REGION Network 2: Watchdog
   // Use S7 comm counter as a live count, but could be anything as long as its changing
   RUNG wire#powerrail
      #Watchdog(bEnable := true, nLocalCount := "S7_Internal_DB".CommCycles, nRemoteCount := "DB_ToHB".WatchdogCounter, sTag := "DB_Customer".Watchdog, bOk => #bWatchdogOk)
   END_RUNG
   // the same network as SCL:
   #Watchdog(bEnable := true,   // "fbHeartbeatCount2"
             nLocalCount := "S7_Internal_DB".CommCycles,
             nRemoteCount := "DB_ToHB".WatchdogCounter,
             sTag := "DB_Customer".Watchdog,
             bOk => #bWatchdogOk);
END_REGION

REGION Network 3: Start request
   RUNG wire#powerrail
      P_Contact(operand := "DB_ToHB".StartRequest, bit := #epStartRequest)
      Contact( "DB_ToHB".EnableHeatbooster )
      S_Coil( "DB_Application".ToHB.StartRequest )
   END_RUNG
   RUNG wire#powerrail
      N_Contact(operand := "DB_ToHB".StartRequest, bit := #enStartRequest)
      R_Coil( "DB_Application".ToHB.StartRequest )
   END_RUNG
   // the same network as SCL:
   #_w1 := "DB_ToHB".StartRequest AND NOT #epStartRequest;   // rising edge of "DB_ToHB".StartRequest
   #epStartRequest := "DB_ToHB".StartRequest;
   IF #_w1 AND "DB_ToHB".EnableHeatbooster THEN "DB_Application".ToHB.StartRequest := TRUE; END_IF;
   #_w2 := NOT "DB_ToHB".StartRequest AND #enStartRequest;   // falling edge of "DB_ToHB".StartRequest
   #enStartRequest := "DB_ToHB".StartRequest;
   IF #_w2 THEN "DB_Application".ToHB.StartRequest := FALSE; END_IF;
END_REGION

REGION Network 4: Stop request
   // a low enable signal is the same as a stop request
   // a watchdog timeout is the same as a stop request
   // a FastStoprequest is also a stop request
   RUNG wire#powerrail
      Contact( "DB_ToHB".StopRequest )
      wire#w1
      Coil( #bStopReq )
   END_RUNG
   RUNG wire#powerrail
      I_Contact( "DB_ToHB".EnableHeatbooster )
   END_RUNG wire#w1
   RUNG wire#powerrail
      I_Contact( #bWatchdogOk )
   END_RUNG wire#w1
   RUNG wire#powerrail
      Contact( "DB_ToHB".FastStopRequest )
   END_RUNG wire#w1
   RUNG wire#powerrail
      P_Contact(operand := #bStopReq, bit := #epStopRequest)
      S_Coil( "DB_Application".ToHB.StopRequest )
   END_RUNG
   RUNG wire#powerrail
      N_Contact(operand := #bStopReq, bit := #enStopRequest)
      R_Coil( "DB_Application".ToHB.StopRequest )
   END_RUNG
   // the same network as SCL:
   #bStopReq := "DB_ToHB".StopRequest OR NOT "DB_ToHB".EnableHeatbooster OR NOT #bWatchdogOk OR "DB_ToHB".FastStopRequest;
   #_w1 := #bStopReq AND NOT #epStopRequest;   // rising edge of #bStopReq
   #epStopRequest := #bStopReq;
   IF #_w1 THEN "DB_Application".ToHB.StopRequest := TRUE; END_IF;
   #_w2 := NOT #bStopReq AND #enStopRequest;   // falling edge of #bStopReq
   #enStopRequest := #bStopReq;
   IF #_w2 THEN "DB_Application".ToHB.StopRequest := FALSE; END_IF;
END_REGION

REGION Network 5: Commands
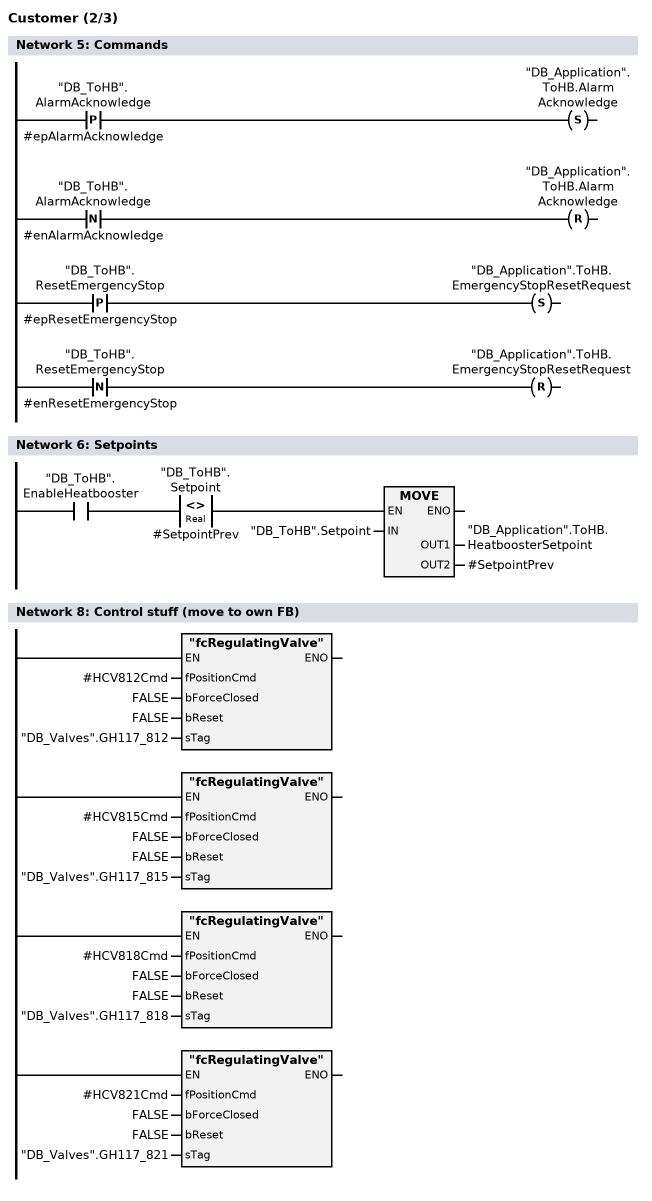
   RUNG wire#powerrail
      P_Contact(operand := "DB_ToHB".AlarmAcknowledge, bit := #epAlarmAcknowledge)
      S_Coil( "DB_Application".ToHB.AlarmAcknowledge )
   END_RUNG
   RUNG wire#powerrail
      N_Contact(operand := "DB_ToHB".AlarmAcknowledge, bit := #enAlarmAcknowledge)
      R_Coil( "DB_Application".ToHB.AlarmAcknowledge )
   END_RUNG
   RUNG wire#powerrail
      P_Contact(operand := "DB_ToHB".ResetEmergencyStop, bit := #epResetEmergencyStop)
      S_Coil( "DB_Application".ToHB.EmergencyStopResetRequest )
   END_RUNG
   RUNG wire#powerrail
      N_Contact(operand := "DB_ToHB".ResetEmergencyStop, bit := #enResetEmergencyStop)
      R_Coil( "DB_Application".ToHB.EmergencyStopResetRequest )
   END_RUNG
   // the same network as SCL:
   #_w1 := "DB_ToHB".AlarmAcknowledge AND NOT #epAlarmAcknowledge;   // rising edge of "DB_ToHB".AlarmAcknowledge
   #epAlarmAcknowledge := "DB_ToHB".AlarmAcknowledge;
   IF #_w1 THEN "DB_Application".ToHB.AlarmAcknowledge := TRUE; END_IF;
   #_w2 := NOT "DB_ToHB".AlarmAcknowledge AND #enAlarmAcknowledge;   // falling edge of "DB_ToHB".AlarmAcknowledge
   #enAlarmAcknowledge := "DB_ToHB".AlarmAcknowledge;
   IF #_w2 THEN "DB_Application".ToHB.AlarmAcknowledge := FALSE; END_IF;
   #_w3 := "DB_ToHB".ResetEmergencyStop AND NOT #epResetEmergencyStop;   // rising edge of "DB_ToHB".ResetEmergencyStop
   #epResetEmergencyStop := "DB_ToHB".ResetEmergencyStop;
   IF #_w3 THEN "DB_Application".ToHB.EmergencyStopResetRequest := TRUE; END_IF;
   #_w4 := NOT "DB_ToHB".ResetEmergencyStop AND #enResetEmergencyStop;   // falling edge of "DB_ToHB".ResetEmergencyStop
   #enResetEmergencyStop := "DB_ToHB".ResetEmergencyStop;
   IF #_w4 THEN "DB_Application".ToHB.EmergencyStopResetRequest := FALSE; END_IF;
END_REGION

REGION Network 6: Setpoints
   RUNG wire#powerrail
      Contact( "DB_ToHB".EnableHeatbooster )
      { S7_Templates := "SrcType := Real" } NE_Contact(in1 := "DB_ToHB".Setpoint, in2 := #SetpointPrev)
      Move(in := "DB_ToHB".Setpoint, out1 => "DB_Application".ToHB.HeatboosterSetpoint, out2 => #SetpointPrev)
   END_RUNG
   // the same network as SCL:
   IF "DB_ToHB".EnableHeatbooster AND ("DB_ToHB".Setpoint <> #SetpointPrev) THEN
       "DB_Application".ToHB.HeatboosterSetpoint := "DB_ToHB".Setpoint;
       #SetpointPrev := "DB_ToHB".Setpoint;
   END_IF;
END_REGION

REGION Network 7 (SCL): To Customer
   "DB_FromHB".CompressorMotorPower            := "DB_Heatbooster".Inverter.HBL_SC_10_A3.fValue;
   "DB_FromHB".CompressorMotorSpeed            := "DB_Heatbooster".Inverter.HBL_SC_10_A1.fValue;
   //"DB_FromHB".HBL_CT_524                      := "DB_Heatbooster".AI.HBL_CT_524.fValue;
   //"DB_FromHB".HBL_CT_538                      := "DB_Heatbooster".AI.HBL_CT_538.fValue;
   "DB_FromHB".HBL_CT_615    := "DB_Heatbooster".AI.HBL_TT_546.fValue;
   "DB_FromHB".HBL_CT_620  := "DB_Heatbooster".AI.HBL_TT_542.fValue;
   "DB_FromHB".HBL_SC_02_A3         := "DB_Heatbooster".AI.HBL_TT_16.fValue;
   "DB_FromHB".HBL_SC_10_A1    := "DB_Heatbooster".AI.HBL_TT_17.fValue;
   "DB_FromHB".HBL_SC_10_A2           := "DB_Heatbooster".AI.HBL_TT_18.fValue;

   "DB_FromHB".HBL_CT_643   := "DB_Heatbooster".AI.HBL_CT_01.fValue;
   "DB_FromHB".HBL_CT_673 := "DB_Heatbooster".AI.HBL_CT_615.fValue;
   "DB_FromHB".HBL_CT_950 := "DB_Heatbooster".AI.HBL_CT_03.fValue;
   "DB_FromHB".HBL_SC_10_A3 := "DB_Heatbooster".AI.SSC_LT_01.fValue;
   "DB_FromHB".TemperatureLift                 := "DB_Heatbooster".Calc.System.TemperatureLift.fValue;
   "DB_FromHB".COP                             := "DB_Heatbooster".Calc.System.COP.fValue;
   "DB_FromHB".HeatSinkHeatRate                := "DB_Heatbooster".Calc.HeatSink.HeatRate.fValue;
   "DB_FromHB".CompressorMotorPower := "DB_Heatbooster".Calc.System.ElectricalPower.fValue;
   "DB_FromHB".HeatboosterPerformance             := "DB_Application".FromHB.HeatboosterSetpoint;
   //"DB_FromHB".WatchdogCounter                := "DB_Application".FromHB.RegulationTarget;
   "DB_FromHB".RunningTimeHours                := INT_TO_UINT("DB_Application".FromHB.RunningTimeHours);
   "DB_FromHB".RunningTimeMinutes              := "DB_Application".FromHB.RunningTimeMinutes;
   "DB_FromHB".RunningTimeSeconds              := "DB_Application".FromHB.RunningTimeSeconds;

   "DB_FromHB".HeatboosterState                := "DB_Application".FromHB.MachineState;
   "DB_FromHB".EmergencyStopStatus             := "DB_Application".FromHB.EmergencyStop;
   "DB_FromHB".HBL_EC_01 := "DB_DO".HBL_EC_01;
   "DB_FromHB".HBL_EC_02 := "DB_DO".HBL_EC_02;
   "DB_FromHB".AlarmActive                    := "DB_DO".GH117_826_1;
   "DB_FromHB".WarningActive                    := "DB_DO".GH117_826_2;

   "DB_FromHB".Alarms                          := "DB_Application".FromHB.Alarms;
   //"DB_FromHB".HBL_SC_03_A1 := FALSE;
   //"DB_FromHB".HBL_SC_03_A2:= FALSE;
   //"DB_FromHB".HBL_SC_03_A3   := FALSE;
   //"DB_FromHB".HBL_SC_01_A1  := FALSE;
   //"DB_FromHB".HBL_SC_01_A2          := 0.0;
   "DB_FromHB".HBL_SC_01_A3            := 0.0;
   "DB_FromHB".HBL_SC_02_A1            := 0.0;
   "DB_FromHB".HBL_SC_02_A2              := 0.0;
   "DB_FromHB".WatchdogCounter                 := "DB_Customer".Watchdog.nLocalCount;
END_REGION

REGION Network 8: Control stuff (move to own FB)
   RUNG wire#powerrail
      "fcRegulatingValve"(fPositionCmd := #HCV812Cmd, bForceClosed := FALSE, bReset := FALSE, sTag := "DB_Valves".GH117_812)
   END_RUNG
   RUNG wire#powerrail
      "fcRegulatingValve"(fPositionCmd := #HCV815Cmd, bForceClosed := FALSE, bReset := FALSE, sTag := "DB_Valves".GH117_815)
   END_RUNG
   RUNG wire#powerrail
      "fcRegulatingValve"(fPositionCmd := #HCV818Cmd, bForceClosed := FALSE, bReset := FALSE, sTag := "DB_Valves".GH117_818)
   END_RUNG
   RUNG wire#powerrail
      "fcRegulatingValve"(fPositionCmd := #HCV821Cmd, bForceClosed := FALSE, bReset := FALSE, sTag := "DB_Valves".GH117_821)
   END_RUNG
   // the same network as SCL:
   "fcRegulatingValve"(fPositionCmd := #HCV812Cmd,
                       bForceClosed := FALSE,
                       bReset := FALSE,
                       sTag := "DB_Valves".GH117_812);
   "fcRegulatingValve"(fPositionCmd := #HCV815Cmd,
                       bForceClosed := FALSE,
                       bReset := FALSE,
                       sTag := "DB_Valves".GH117_815);
   "fcRegulatingValve"(fPositionCmd := #HCV818Cmd,
                       bForceClosed := FALSE,
                       bReset := FALSE,
                       sTag := "DB_Valves".GH117_818);
   "fcRegulatingValve"(fPositionCmd := #HCV821Cmd,
                       bForceClosed := FALSE,
                       bReset := FALSE,
                       sTag := "DB_Valves".GH117_821);
END_REGION

REGION Network 9: Analog outputs
   // Move to own FB in Section 30
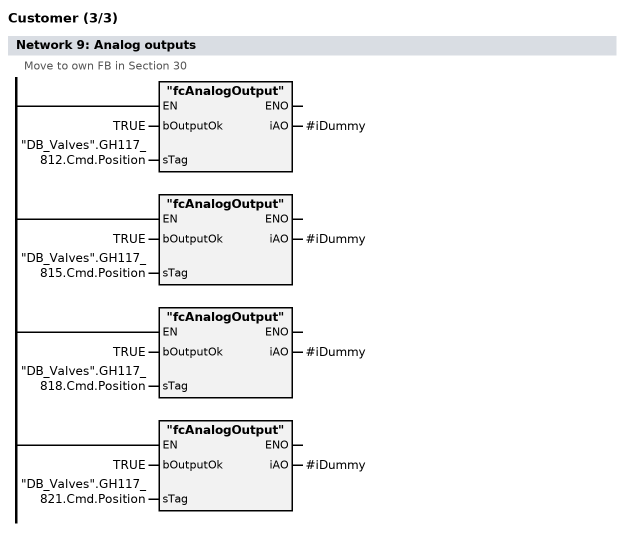
   RUNG wire#powerrail
      "fcAnalogOutput"(bOutputOk := TRUE, sTag := "DB_Valves".GH117_812.Cmd.Position, iAO => #iDummy)
   END_RUNG
   RUNG wire#powerrail
      "fcAnalogOutput"(bOutputOk := TRUE, sTag := "DB_Valves".GH117_815.Cmd.Position, iAO => #iDummy)
   END_RUNG
   RUNG wire#powerrail
      "fcAnalogOutput"(bOutputOk := TRUE, sTag := "DB_Valves".GH117_818.Cmd.Position, iAO => #iDummy)
   END_RUNG
   RUNG wire#powerrail
      "fcAnalogOutput"(bOutputOk := TRUE, sTag := "DB_Valves".GH117_821.Cmd.Position, iAO => #iDummy)
   END_RUNG
   // the same network as SCL:
   "fcAnalogOutput"(bOutputOk := TRUE, sTag := "DB_Valves".GH117_812.Cmd.Position, iAO => #iDummy);
   "fcAnalogOutput"(bOutputOk := TRUE, sTag := "DB_Valves".GH117_815.Cmd.Position, iAO => #iDummy);
   "fcAnalogOutput"(bOutputOk := TRUE, sTag := "DB_Valves".GH117_818.Cmd.Position, iAO => #iDummy);
   "fcAnalogOutput"(bOutputOk := TRUE, sTag := "DB_Valves".GH117_821.Cmd.Position, iAO => #iDummy);
END_REGION
END_FUNCTION_BLOCK

FUNCTION "fcCustomerMapping" : Void   // FC1, FBD
TITLE = Map IO tags to DBs
{ S7_Optimized_Access := 'TRUE' }
VERSION : 0.1
// stored: AutoNumber true, IsIECCheckEnabled false, SetENOAutomatically false, UDAEnableTagReadback false
BEGIN

REGION Network 1 (SCL): Comments
   // If using S7 communication with the customer, use DB_ToHB & DB_FromHB
   // If not, still move everything into these DBs, but then use this block for copying to/from I/O memory
   // Also, the DBs can contain a superset of those things actually sent or received (S7 communication has higher bandwidth)
   // Could also be in its own OB, just like Modbus, so it can "feed into" DB_ToHB and DB_FromHB transparently
END_REGION

REGION Network 2 (SCL): Signals in from customer ("ToHb")
   // Commands
   //"DB_ToHB".StartRequest := "VB3-M8301 Start";

   // Customer-specific signals
   //"DB_ToHB".Setpoint := "ScaleIn"(nIn := "QI117_828B1");
END_REGION

REGION Network 3 (SCL): Signals out to Customer ("FromHB")
   // Status bits
   //"VB3-M8301 NA-Status"   := "DB_FromHB".EmergencyStopStatus;
END_REGION
END_FUNCTION

FUNCTION "fcRegulatingValve" : Void
{ S7_Optimized_Access := 'TRUE' }
VERSION : 0.1
   VAR_INPUT 
      fPositionCmd : Real;
      bForceClosed : Bool;   // 1 = force closed, 0 = do not force closed
      bReset : Bool;   // 1 = reset manual mode
   END_VAR

   VAR_IN_OUT 
      sTag : "stRegulatingValve";
   END_VAR


BEGIN
	// Regulating valve
	
	// Reset manual mode
	IF #bReset THEN
	    #sTag.Cmd.bManualMode := FALSE;
	    #sTag.Cmd.fManualValue := 0.0;
	END_IF;
	
	IF #sTag.Cmd.bManualMode = TRUE THEN
	    #sTag.Cmd.Position.Eng.fValue := #sTag.Cmd.fManualValue;
	ELSIF #bForceClosed = TRUE THEN
	    #sTag.Cmd.Position.Eng.fValue := #sTag.Cmd.fOffset;
	ELSIF #sTag.Cmd.fOffset = 0.0 THEN
	    #sTag.Cmd.Position.Eng.fValue := #fPositionCmd;
	ELSE
	    // squeeze [fMin,fMax] into the range [fOffset,fMax] to account for a nonzero closed position but still reach fully open at 100%
	    #sTag.Cmd.Position.Eng.fValue := "fcRescale"(InMin := #sTag.Cmd.Position.Eng.fMin, 
	                                                InMax  := #sTag.Cmd.Position.Eng.fMax,
	                                                InVal  := #fPositionCmd,
	                                                OutMin := #sTag.Cmd.fOffset,
	                                                OutMax := #sTag.Cmd.Position.Eng.fMax);
	END_IF;
END_FUNCTION

FUNCTION "fcRescale" : Real
{ S7_Optimized_Access := 'TRUE' }
VERSION : 0.1
   VAR_INPUT 
      InMin : Real;
      InMax : Real;
      InVal : Real;
      OutMin : Real;
      OutMax : Real;
   END_VAR


BEGIN
	// Real-to-real rescaling of a value
	
	#fcRescale := #OutMax - ((#OutMax - #OutMin) / (#InMax - #InMin)) * (#InMax - #InVal);
END_FUNCTION

FUNCTION "fcAnalogOutput" : Void
{ S7_Optimized_Access := 'TRUE' }
VERSION : 0.1
   VAR_INPUT 
      bOutputOk : Bool;   // 1 = output channel/module/fieldbus device is working, 0 = not working
   END_VAR

   VAR_OUTPUT 
      iAO : Int;   // Raw value to write
   END_VAR

   VAR_IN_OUT 
      sTag : "stAnalogOutput";   // Output channel scaling parameters
   END_VAR

   VAR_TEMP 
      fSlope : Real;
      iIntercept : Int;
   END_VAR


BEGIN
	// Scale a CalcValue to a raw value
	
	// Output channel status. Scale always even if output channel is not ok
	#sTag.Raw.bFault := NOT(#bOutputOk);
	// Scaling. Only intervene if the value is invalid or NaN
	IF #sTag.Eng.bError = TRUE OR "isNaN"(#sTag.Eng.fValue) THEN
	    #sTag.Raw.iValue := 0;
	ELSE
	    // NOTE: not detecting division by zero here
	    #fSlope := INT_TO_REAL(#sTag.Raw.iMax - #sTag.Raw.iMin) / (#sTag.Eng.fMax - #sTag.Eng.fMin);
	    #iIntercept := #sTag.Raw.iMax - REAL_TO_INT(#fSlope * #sTag.Eng.fMax);
	    #sTag.Raw.iValue := REAL_TO_INT(#sTag.Eng.fValue*#fSlope) + #iIntercept;
	END_IF;
	
	// Local outputs
	#iAO := #sTag.Raw.iValue;
END_FUNCTION

FUNCTION "isNaN" : Bool   // FC19, FBD
TITLE = isNaN
{ S7_Optimized_Access := 'TRUE' }
VERSION : 0.1
// Returns TRUE if a REAL is NaN
// stored: AutoNumber true, IsIECCheckEnabled false, SetENOAutomatically false, UDAEnableTagReadback false
   VAR_INPUT
      In : Real;
   END_VAR
BEGIN

REGION Network 1
   // NOT_OK is a compiler builtin, but not available in SCL
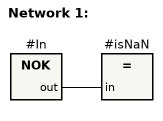
   // no SCL statement known for NOK: written as a call
   #isNaN := NOK(#In);
END_REGION
END_FUNCTION

FUNCTION_BLOCK "Cloud"   // FB4, FBD
TITLE = Cloud tasks
{ S7_Optimized_Access := 'TRUE' }
VERSION : 0.1
// stored: AutoNumber true, IsIECCheckEnabled false, IsRetainMemResEnabled false, MemoryReserve 0, SetENOAutomatically false, UDAEnableTagReadback false
   VAR
      CurrentTime { ExternalWritable := 'False'} : DTL;
      SetTime : DTL;
      Update : Bool;
   END_VAR
   VAR_TEMP
      ReadStatus : Int;
      WriteStatus : Int;
   END_VAR
   VAR_TEMP   // added for the SCL form of the ladder/FBD networks
      _w1 : Bool;
   END_VAR
BEGIN

REGION Network 1: Read PLC clock
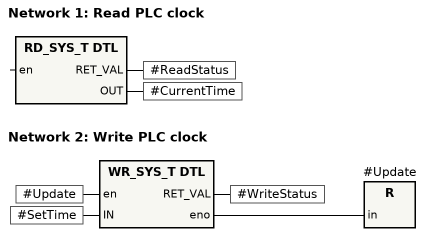
   #ReadStatus := RD_SYS_T(OUT => #CurrentTime);
END_REGION

REGION Network 2: Write PLC clock
   #WriteStatus := WR_SYS_T(EN := #Update, IN := #SetTime, ENO => #_w1);
   IF #_w1 THEN #Update := FALSE; END_IF;
END_REGION

REGION Network 3 (SCL): Manually copy interesting values to its own DB
   // This prevents messing up OPC UA URIs every time something unrelated in the program changes
   // AI
   "DB_Cloud".HBL_TT_502 := "DB_Heatbooster".AI.HBL_TT_502.fValue;
   "DB_Cloud".HBL_PT_503 := "DB_Heatbooster".AI.HBL_PT_503.fValue;
   "DB_Cloud".HBL_TT_504 := "DB_Heatbooster".AI.HBL_TT_504.fValue;
   "DB_Cloud".HBL_LT_510 := "DB_Heatbooster".AI.HBL_LT_510.fValue;
   "DB_Cloud".HBL_PT_511 := "DB_Heatbooster".AI.HBL_PT_511.fValue;
   "DB_Cloud".HBL_TT_512 := "DB_Heatbooster".AI.HBL_TT_512.fValue;
   "DB_Cloud".HBL_TT_516 := "DB_Heatbooster".AI.HBL_TT_516.fValue;
   "DB_Cloud".HBL_PT_517 := "DB_Heatbooster".AI.HBL_PT_517.fValue;
   "DB_Cloud".HBL_TT_518 := "DB_Heatbooster".AI.HBL_TT_518.fValue;
   "DB_Cloud".HBL_PT_519 := "DB_Heatbooster".AI.HBL_PT_519.fValue;
   "DB_Cloud".HBL_FT_520 := "DB_Heatbooster".AI.HBL_FT_520.fValue;
   "DB_Cloud".HBL_TT_530 := "DB_Heatbooster".AI.HBL_TT_530.fValue;
   "DB_Cloud".HBL_PT_531 := "DB_Heatbooster".AI.HBL_PT_531.fValue;
   "DB_Cloud".HBL_TT_532 := "DB_Heatbooster".AI.HBL_TT_532.fValue;
   "DB_Cloud".HBL_TT_533 := "DB_Heatbooster".AI.HBL_TT_533.fValue;
   "DB_Cloud".HBL_PT_534 := "DB_Heatbooster".AI.HBL_PT_534.fValue;
   "DB_Cloud".HBL_AT_535 := "DB_Heatbooster".AI.HBL_AT_535.fValue;
   "DB_Cloud".HBL_TT_540 := "DB_Heatbooster".AI.HBL_TT_540.fValue;
   "DB_Cloud".HBL_PT_541 := "DB_Heatbooster".AI.HBL_PT_541.fValue;
   "DB_Cloud".HBL_TT_542 := "DB_Heatbooster".AI.HBL_TT_542.fValue;
   "DB_Cloud".HBL_TT_543 := "DB_Heatbooster".AI.HBL_TT_543.fValue;
   "DB_Cloud".HBL_PT_544 := "DB_Heatbooster".AI.HBL_PT_544.fValue;
   "DB_Cloud".HBL_AT_545 := "DB_Heatbooster".AI.HBL_AT_545.fValue;
   "DB_Cloud".HBL_TT_546 := "DB_Heatbooster".AI.HBL_TT_546.fValue;
   "DB_Cloud".HBL_PT_547 := "DB_Heatbooster".AI.HBL_PT_547.fValue;
   "DB_Cloud".HBL_TT_571 := "DB_Heatbooster".AI.HBL_TT_571.fValue;
   "DB_Cloud".HBL_PT_572 := "DB_Heatbooster".AI.HBL_PT_572.fValue;
   "DB_Cloud".HBL_TT_573 := "DB_Heatbooster".AI.HBL_TT_573.fValue;
   "DB_Cloud".HBL_LT_610 := "DB_Heatbooster".AI.HBL_LT_610.fValue;
   "DB_Cloud".HBL_TT_611 := "DB_Heatbooster".AI.HBL_TT_611.fValue;
   "DB_Cloud".HBL_PT_612 := "DB_Heatbooster".AI.HBL_PT_612.fValue;
   "DB_Cloud".HBL_CT_615 := "DB_Heatbooster".AI.HBL_CT_615.fValue;
   "DB_Cloud".HBL_PT_618 := "DB_Heatbooster".AI.HBL_PT_618.fValue;
   "DB_Cloud".HBL_PT_635 := "DB_Heatbooster".AI.HBL_PT_635.fValue;
   "DB_Cloud".HBL_PT_636 := "DB_Heatbooster".AI.HBL_PT_636.fValue;
   "DB_Cloud".HBL_LT_650 := "DB_Heatbooster".AI.HBL_LT_650.fValue;
   "DB_Cloud".HBL_PT_651 := "DB_Heatbooster".AI.HBL_PT_651.fValue;
   "DB_Cloud".HBL_PT_701 := "DB_Heatbooster".AI.HBL_PT_701.fValue;
   "DB_Cloud".HBL_PT_702 := "DB_Heatbooster".AI.HBL_PT_702.fValue;
   "DB_Cloud".HBL_PT_703 := "DB_Heatbooster".AI.HBL_PT_703.fValue;
   "DB_Cloud".CPC_LT_870 := "DB_Heatbooster".AI.CPC_LT_870.fValue;
   "DB_Cloud".CPC_TT_871 := "DB_Heatbooster".AI.CPC_TT_871.fValue;
   "DB_Cloud".CPC_PT_872 := "DB_Heatbooster".AI.CPC_PT_872.fValue;
   "DB_Cloud".CPC_PT_862 := "DB_Heatbooster".AI.CPC_PT_862.fValue;
   "DB_Cloud".HBL_TT_901 := "DB_Heatbooster".AI.HBL_TT_901.fValue;
   "DB_Cloud".HBL_PT_902 := "DB_Heatbooster".AI.HBL_PT_902.fValue;
   "DB_Cloud".HBL_TT_03  := "DB_Heatbooster".AI.HBL_TT_03.fValue;
   "DB_Cloud".HBL_TT_16  := "DB_Heatbooster".AI.HBL_TT_16.fValue;
   "DB_Cloud".HBL_TT_17  := "DB_Heatbooster".AI.HBL_TT_17.fValue;
   "DB_Cloud".HBL_TT_18  := "DB_Heatbooster".AI.HBL_TT_18.fValue;
   "DB_Cloud".HBL_TT_20  := "DB_Heatbooster".AI.HBL_TT_20.fValue;
   "DB_Cloud".HBL_TT_21  := "DB_Heatbooster".AI.HBL_TT_21.fValue;
   "DB_Cloud".HBL_TT_22  := "DB_Heatbooster".AI.HBL_TT_22.fValue;
   "DB_Cloud".HBL_TT_23  := "DB_Heatbooster".AI.HBL_TT_23.fValue;
   "DB_Cloud".HBL_TT_24  := "DB_Heatbooster".AI.HBL_TT_24.fValue;
   "DB_Cloud".HBL_TT_25  := "DB_Heatbooster".AI.HBL_TT_25.fValue;
   "DB_Cloud".HBL_TT_26  := "DB_Heatbooster".AI.HBL_TT_26.fValue;
   "DB_Cloud".HBL_TT_27  := "DB_Heatbooster".AI.HBL_TT_27.fValue;
   "DB_Cloud".HBL_PT_05  := "DB_Heatbooster".AI.HBL_PT_05.fValue;
   "DB_Cloud".HBL_PT_06  := "DB_Heatbooster".AI.HBL_PT_06.fValue;
   "DB_Cloud".HBL_PT_17  := "DB_Heatbooster".AI.HBL_PT_17.fValue;
   "DB_Cloud".HBL_CT_01  := "DB_Heatbooster".AI.HBL_CT_01.fValue;
   "DB_Cloud".HBL_CT_03  := "DB_Heatbooster".AI.HBL_CT_03.fValue;
   "DB_Cloud".SSC_TT_01  := "DB_Heatbooster".AI.SSC_TT_01.fValue;
   "DB_Cloud".SSC_TT_02  := "DB_Heatbooster".AI.SSC_TT_02.fValue;
   "DB_Cloud".SSC_TT_03  := "DB_Heatbooster".AI.SSC_TT_03.fValue;
   "DB_Cloud".SSC_TT_04  := "DB_Heatbooster".AI.SSC_TT_04.fValue;
   "DB_Cloud".SSC_PIT_01 := "DB_Heatbooster".AI.SSC_PIT_01.fValue;
   "DB_Cloud".SSC_PDT_01 := "DB_Heatbooster".AI.SSC_PDT_01.fValue;
   "DB_Cloud".SSC_LT_01  := "DB_Heatbooster".AI.SSC_LT_01.fValue;
   "DB_Cloud".HBL_VT_01 := "DB_Heatbooster".AI.HBL_VT_01.fValue;
   "DB_Cloud".HBL_TT_36 := "DB_Heatbooster".AI.HBL_TT_36.fValue;

   // Calc
   "DB_Cloud".Compressor_CrankcaseSaturationTemperature := "DB_Heatbooster".Calc.Compressor.CrankcaseSaturationTemperature.fValue;
   "DB_Cloud".Compressor_CrankcaseSuperheat := "DB_Heatbooster".Calc.Compressor.CrankcaseSuperheat.fValue;
   "DB_Cloud".Compressor_VolumetricEfficiency := "DB_Heatbooster".Calc.Compressor.VolumetricEfficiency.fValue;
   "DB_Cloud".Compressor_IsentropicEfficiency := "DB_Heatbooster".Calc.Compressor.IsentropicEfficiency.fValue;
   "DB_Cloud".Compressor_Massflow := "DB_Heatbooster".Calc.Compressor.Massflow.fValue;
   "DB_Cloud".HeatSink_DeltaT := "DB_Heatbooster".Calc.HeatSink.DeltaT.fValue;
   "DB_Cloud".HeatSink_Pinch := "DB_Heatbooster".Calc.HeatSink.Pinch.fValue;
   "DB_Cloud".HeatSink_HeatRate := "DB_Heatbooster".Calc.HeatSink.HeatRate.fValue;
   "DB_Cloud".HeatSink_DeltaP := "DB_Heatbooster".Calc.HeatSink.DeltaP.fValue;
   "DB_Cloud".HeatSink_Massflow := "DB_Heatbooster".Calc.HeatSink.Massflow.fValue;
   "DB_Cloud".HeatSource_DeltaT := "DB_Heatbooster".Calc.HeatSource.DeltaT.fValue;
   "DB_Cloud".HeatSource_Pinch := "DB_Heatbooster".Calc.HeatSource.Pinch.fValue;
   "DB_Cloud".HeatSource_HeatRate := "DB_Heatbooster".Calc.HeatSource.HeatRate.fValue;
   "DB_Cloud".HeatSource_DeltaP := "DB_Heatbooster".Calc.HeatSource.DeltaP.fValue;
   "DB_Cloud".HeatSource_TemperatureRateOfChange := "DB_Heatbooster".Calc.HeatSource.TemperatureRateOfChange.fValue;
   "DB_Cloud".HeatSource_Massflow := "DB_Heatbooster".Calc.HeatSource.Massflow.fValue;
   "DB_Cloud".HighPressPart_CompressorSaturationTemperature := "DB_Heatbooster".Calc.HighPressPart.CompressorSaturationTemperature.fValue;
   "DB_Cloud".HighPressPart_CompressorSuperheat := "DB_Heatbooster".Calc.HighPressPart.CompressorSuperheat.fValue;
   "DB_Cloud".HighPressPart_CondenserSaturationTemperature := "DB_Heatbooster".Calc.HighPressPart.CondenserSaturationTemperature.fValue;
   "DB_Cloud".HighPressPart_CondenserSubcooling := "DB_Heatbooster".Calc.HighPressPart.CondenserSubcooling.fValue;
   "DB_Cloud".HighPressPart_ExpansionValveSubcooling := "DB_Heatbooster".Calc.HighPressPart.ExpansionValveSubcooling.fValue;
   "DB_Cloud".HighPressPart_CondenserDeltaP := "DB_Heatbooster".Calc.HighPressPart.CondenserDeltaP.fValue;
   "DB_Cloud".LowPressPart_EvaporatorSuperheat := "DB_Heatbooster".Calc.LowPressPart.EvaporatorSuperheat.fValue;
   "DB_Cloud".LowPressPart_CompressorSuperheat := "DB_Heatbooster".Calc.LowPressPart.CompressorSuperheat.fValue;
   "DB_Cloud".LowPressPart_EvaporatorSaturationTemperature := "DB_Heatbooster".Calc.LowPressPart.EvaporatorSaturationTemperature.fValue;
   "DB_Cloud".LowPressPart_CompressorSaturationTemperature := "DB_Heatbooster".Calc.LowPressPart.CompressorSaturationTemperature.fValue;
   "DB_Cloud".System_Quality := "DB_Heatbooster".Calc.System.Quality.fValue;
   "DB_Cloud".System_COP := "DB_Heatbooster".Calc.System.COP.fValue;
   "DB_Cloud".System_ElectricalPower := "DB_Heatbooster".Calc.System.ElectricalPower.fValue;
   "DB_Cloud".System_TemperatureLift := "DB_Heatbooster".Calc.System.TemperatureLift.fValue;
   "DB_Cloud".System_MotorEfficiency := "DB_Heatbooster".Calc.System.MotorEfficiency.fValue;
   "DB_Cloud".System_FMEP := "DB_Heatbooster".Calc.System.FMEP.fValue;
   "DB_Cloud".Auxiliary_ShaftSealDeltaT := "DB_Heatbooster".Calc.Auxiliary.ShaftSealDeltaT.fValue;
   "DB_Cloud".Auxiliary_CPCPumpDeltaP := "DB_Heatbooster".Calc.Auxiliary.CPCPumpDeltaP.fValue;
   "DB_Cloud".Misc_OilFilterDeltaP := "DB_Heatbooster".Calc.Misc.OilFilterDeltaP.fValue;

   // DI
   "DB_Cloud".HBL_FS_01 := "DB_Heatbooster".DI.HBL_FS_01;
   "DB_Cloud".HBL_FS_02 := "DB_Heatbooster".DI.HBL_FS_02;
   "DB_Cloud".HBL_LS_632 := "DB_Heatbooster".DI.HBL_LS_632;
   "DB_Cloud".HBL_LS_633 := "DB_Heatbooster".DI.HBL_LS_633;
   "DB_Cloud".CPC_LS_864 := "DB_Heatbooster".DI.CPC_LS_864;
   "DB_Cloud".VPNUserConnected := "DB_Heatbooster".DI.VPNUserConnected;

   // DO
   "DB_Cloud".HBL_EC_01 := "DB_Heatbooster".DO.HBL_EC_01;
   "DB_Cloud".HBL_EC_02 := "DB_Heatbooster".DO.HBL_EC_02;
   "DB_Cloud".HBL_HV_630 := "DB_Heatbooster".DO.HBL_HV_630;
   "DB_Cloud".HBL_HV_631 := "DB_Heatbooster".DO.HBL_HV_631;
   "DB_Cloud".HBL_HV_860 := "DB_Heatbooster".DO.HBL_HV_860;
   "DB_Cloud".HBL_HV_861 := "DB_Heatbooster".DO.HBL_HV_861;
   "DB_Cloud".SSC_P_01 := "DB_Heatbooster".DO.SSC_P_01;
   "DB_Cloud".SSC_F_01 := "DB_Heatbooster".DO.SSC_F_01;
   "DB_Cloud".SSC_P_02 := "DB_Heatbooster".DO.SSC_P_02;
   "DB_Cloud".CPC_P_01 := "DB_Heatbooster".DO.CPC_P_01;

   // Inverter
   "DB_Cloud".HBL_SC_01_A1 := "DB_Heatbooster".Inverter.HBL_SC_01_A1.fValue;
   "DB_Cloud".HBL_SC_01_A2 := "DB_Heatbooster".Inverter.HBL_SC_01_A2.fValue;
   "DB_Cloud".HBL_SC_01_A3 := "DB_Heatbooster".Inverter.HBL_SC_01_A3.fValue;
   "DB_Cloud".HBL_SC_02_A1 := "DB_Heatbooster".Inverter.HBL_SC_02_A1.fValue;
   "DB_Cloud".HBL_SC_02_A2 := "DB_Heatbooster".Inverter.HBL_SC_02_A2.fValue;
   "DB_Cloud".HBL_SC_02_A3 := "DB_Heatbooster".Inverter.HBL_SC_02_A3.fValue;
   "DB_Cloud".HBL_SC_03_A1 := "DB_Heatbooster".Inverter.HBL_SC_03_A1.fValue;
   "DB_Cloud".HBL_SC_03_A2 := "DB_Heatbooster".Inverter.HBL_SC_03_A2.fValue;
   "DB_Cloud".HBL_SC_03_A3 := "DB_Heatbooster".Inverter.HBL_SC_03_A3.fValue;
   "DB_Cloud".HBL_SC_10_A1 := "DB_Heatbooster".Inverter.HBL_SC_10_A1.fValue;
   "DB_Cloud".HBL_SC_10_A2 := "DB_Heatbooster".Inverter.HBL_SC_10_A2.fValue;
   "DB_Cloud".HBL_SC_10_A3 := "DB_Heatbooster".Inverter.HBL_SC_10_A3.fValue;

   // Valves
   "DB_Cloud".HBL_HCV_576_A1 := "DB_Heatbooster".Valve.HBL_HCV_576_A1.fValue;
   "DB_Cloud".HBL_HCV_578_A1 := "DB_Heatbooster".Valve.HBL_HCV_578_A1.fValue;
   "DB_Cloud".HBL_HCV_577_A1 := "DB_Heatbooster".Valve.HBL_HCV_577_A1.fValue;
   "DB_Cloud".HBL_HCV_579_A1 := "DB_Heatbooster".Valve.HBL_HCV_579_A1.fValue;
   "DB_Cloud".HBL_HCV_515_A1 := "DB_Heatbooster".Valve.HBL_HCV_515_A1.fValue;
   "DB_Cloud".HBL_HCV_575_A1 := "DB_Heatbooster".Valve.HBL_HCV_575_A1.fValue;
   "DB_Cloud".HBL_HCV_616_A1 := "DB_Heatbooster".Valve.HBL_HCV_616_A1.fValue;
   "DB_Cloud".HBL_HCV_700_A1 := "DB_Heatbooster".Valve.HBL_HCV_700_A1.fValue;
   "DB_Cloud".HBL_HCV_514_A1 := "DB_Heatbooster".Valve.HBL_HCV_514_A1.fValue;
   "DB_Cloud".HBL_HCV_548_A1 := "DB_Heatbooster".Valve.HBL_HCV_548_A1.fValue;

   // Other
   "DB_Cloud".ClientID := "DB_System".ClientID;
   "DB_Cloud".RunningTimeHours := "DB_Application".FromHB.RunningTimeHours;
   "DB_Cloud".RunningTimeMinutes := "DB_Application".FromHB.RunningTimeMinutes;
   "DB_Cloud".RunningTimeSeconds := "DB_Application".FromHB.RunningTimeSeconds;
   "DB_Cloud".MachineState := "DB_Application".FromHB.MachineState;
END_REGION
END_FUNCTION_BLOCK

FUNCTION "SoftwareVersion" : String
{ S7_Optimized_Access := 'TRUE' }
AUTHOR : Heaten
VERSION : 0.1

BEGIN
	// SOFTWARE VERSION: in-band software change tracking
	// Changes and descriptions are usually tracked out-of-band, eg as git commit messages or as issues in github etc. This is to more tightly couple change tracking with the actual project.
	// INSTRUCTIONS:
	// 1. New entries should go at the top, such that the most recent changes are visible first.
	// 2. Be short but descriptive; one line per change is a good starting point.
	// 3. Change the version number. This is a string so there is a lot of flexibility as to the format.
	
	#SoftwareVersion := 'V5.0.1.1';
	
	// V5.0.1.1
	// Added customer variables to DB_ToHB to be able to compile software
	// Changes in Process_PLC
	
	// V5.0.1.0 Changes in HMI and Process_PLC
	
	// V5.0.0.0 26.02.2025
	// - forked from Alpha-2 V4.0.0.7
	// - V5 is for the split-system steam/steam
	
END_FUNCTION

ORGANIZATION_BLOCK "CAN_CyclicInterrupt"   // OB30, FBD, CyclicInterrupt
{ S7_Optimized_Access := 'TRUE' }
VERSION : 0.1
// stored: AutoNumber true, IsIECCheckEnabled false, SetENOAutomatically false
   VAR_INPUT
      Initial_Call : Bool;   // Initial call of this OB
      Event_Count : Int;   // Events discarded
   END_VAR
BEGIN

REGION Network 1: CAN communication
   // EN := "DB_CurrentSetting"."CAN-Module_Active"
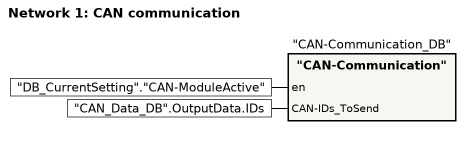
   IF "DB_CurrentSetting"."CAN-ModuleActive" THEN
       "CAN-Communication_DB"("CAN-IDs_ToSend" := "CAN_Data_DB".OutputData.IDs);   // "CAN-Communication"
   END_IF;
END_REGION
END_ORGANIZATION_BLOCK

FUNCTION_BLOCK "CAN-Communication"   // FB8, FBD
{ S7_Optimized_Access := 'TRUE' }
VERSION : 0.1
// stored: AutoNumber true, IsIECCheckEnabled false, IsRetainMemResEnabled false, MemoryReserve 100, SetENOAutomatically false, UDAEnableTagReadback false
   VAR_IN_OUT
      "CAN-IDs_ToSend" : Array[0..74] of Int;
   END_VAR
   VAR
      SendBusy : Bool;
      UseFixedPoint : Bool;   // Send data on CAN as fixed point
      Memory : DInt;
      CycleCheck : Bool;
      TESTUINT_CTRL { ExternalAccessible := 'False'; ExternalVisible := 'False'; ExternalWritable := 'False'} : UInt;
      TESTUINT_SEND : UInt;
      TESTUINT_RCV : UInt;
      TOF_SendError { S7_SetPoint := 'True'} : TOF_TIME;
      CountSendAll : UDInt;
      ScaleFactor : Real := 1000.0;   // Fixed point scale factor
   END_VAR
   VAR_TEMP
      i : Int;
      UpperBound : DInt;
      NumberOfFrames : SInt;
      TestUint : UInt;
   END_VAR
BEGIN

REGION Network 1: CAN Control
   // process a CAN_CTRL command (if requested)
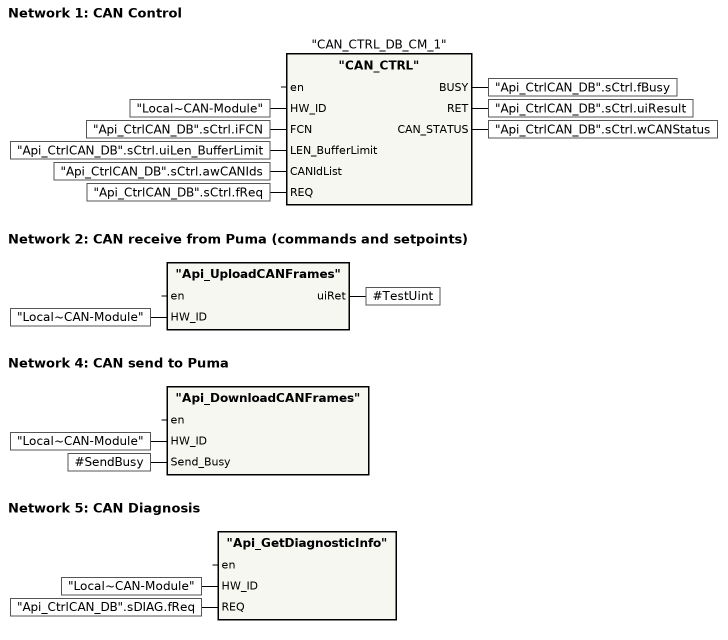
   "CAN_CTRL_DB_CM_1"(HW_ID := "Local~CAN-Module",   // "CAN_CTRL"
                      FCN := "Api_CtrlCAN_DB".sCtrl.iFCN,
                      LEN_BufferLimit := "Api_CtrlCAN_DB".sCtrl.uiLen_BufferLimit,
                      CANIdList := "Api_CtrlCAN_DB".sCtrl.awCANIds,
                      REQ := "Api_CtrlCAN_DB".sCtrl.fReq,
                      BUSY => "Api_CtrlCAN_DB".sCtrl.fBusy,
                      RET => "Api_CtrlCAN_DB".sCtrl.uiResult,
                      CAN_STATUS => "Api_CtrlCAN_DB".sCtrl.wCANStatus);
END_REGION

REGION Network 2: CAN receive from Puma (commands and setpoints)
   // function processes the upload of CAN frames and processes the uploaded CAN frames
   "Api_UploadCANFrames"(HW_ID := "Local~CAN-Module", uiRet => #TestUint);
END_REGION

REGION Network 3 (SCL): Send CAN frame select
   // The CAN SEND block can only send 19 frames each call. So every call, other frame IDs gets written into the output list.
   // HW_ID := "Local~CAN-Module"
   //Diagnosis to store error messages from CAN functions
   IF "Api_CtrlCAN_DB".sCtrl.uiResult <> 0 THEN
       #TESTUINT_CTRL:="Api_CtrlCAN_DB".sCtrl.uiResult;
   END_IF;
   IF "Api_CtrlCAN_DB".sSEND.sDemo.sDownload.uiResult <> 0 THEN
       #TESTUINT_SEND:="Api_CtrlCAN_DB".sSEND.sDemo.sDownload.uiResult;
   END_IF;
   IF #TestUint <> 0 THEN
       #TESTUINT_RCV := #TestUint;
   END_IF;

   IF NOT "Api_CtrlCAN_DB".sRCV.fReq THEN // Was ist das und wofür?
       "Api_CtrlCAN_DB".sCtrl.fReq := True;
       "Api_CtrlCAN_DB".sCtrl.iFCN := 1;
       "Api_CtrlCAN_DB".sRCV.fReq := True;
   END_IF;


   //Update current status
   IF "Api_CtrlCAN_DB".sSEND.fTransfer AND #SendBusy THEN //If completed transmission pending then check current status
       "Api_DownloadCANFrames"(HW_ID := "Local~CAN-Module",
                               Send_Busy := #SendBusy);
   END_IF; // "Api_CtrlCAN_DB".sSEND.fTransfer THEN 

   //Write IDs to send list
   IF NOT "Api_CtrlCAN_DB".sSEND.fTransfer AND NOT #SendBusy THEN // OR NOT "Api_CtrlCAN_DB".sSEND.sDemo.sRequest.fReq THEN
       // In Transfere is ready or actually no send request (first or due to error)    
       // Currently in case of error we do not resend this on, but proceed with the other ones. It is only retransmitted within the normal procedure after a complete cycle.
       // "Api_CtrlCAN_DB".sSEND.sDemo.sRequest.fError ist die error flag

       //#UpperBound := UPPER_BOUND(ARR := #"CAN-IDs_ToSend", DIM := 1);     //Upper bound of all CAN-IDs to send
       #UpperBound := 69;
       #NumberOfFrames := 0;                                               //Resetting CAN frame counter
       FOR #i := 0 TO 18 DO                                                //Writing all 10/19 CAN_IDs to send into output array
           IF #Memory + #i <= #UpperBound THEN                             //Check if there are CAN-IDs left
               "Api_CtrlCAN_DB".sSEND.sDemo.sRequest.aiCAN_ID[#i] := #"CAN-IDs_ToSend"[#i + #Memory];      //The next ID gets written into send list
               #NumberOfFrames := #NumberOfFrames + 1;                     //Count up on each frame
           ELSE
               "Api_CtrlCAN_DB".sSEND.sDemo.sRequest.aiCAN_ID[#i] := 0;    //No ID left
           END_IF;

       END_FOR;

       "Api_CtrlCAN_DB".sSEND.sDemo.sRequest.siNoFrames := #NumberOfFrames;//Send number of CAN-IDs to send to maximum (19 [0..18])
       "Api_CtrlCAN_DB".sSEND.sDemo.sRequest.fReq := TRUE;                 //send new frame if not busy

       #Memory := #Memory + #NumberOfFrames;                               //Next cycle the Next 19 IDs gets send 
       IF #Memory > #UpperBound THEN   //if all IDs got send, all gets send again
           #Memory := 0;               //Start with ID 0
           #CountSendAll += 1;
       END_IF; // IF #Memory > #UpperBound THEN

   END_IF; // IF NOT "Api_CtrlCAN_DB".sSEND.fTransfer OR NOT "Api_CtrlCAN_DB".sSEND.sDemo.sRequest.fReq THEN
END_REGION

REGION Network 4: CAN send to Puma
   // function checks if CAN frames shall be transitted, which CAN frames shall be transmitted, enters the requested CAN frames in the data field that will be written to the CM module and processes the download to the CM module
   "Api_DownloadCANFrames"(HW_ID := "Local~CAN-Module", Send_Busy := #SendBusy);
END_REGION

REGION Network 5: CAN Diagnosis
   // process "Get Diagnostic Information" (if requested)
   "Api_GetDiagnosticInfo"(HW_ID := "Local~CAN-Module", REQ := "Api_CtrlCAN_DB".sDIAG.fReq);
END_REGION

REGION Network 6: Error message via CAN
   // WinCC Alarm 3001 triggered from:
   // "CAN_Data_DB".InputData.CAN_ID_101h.Error_CAN
   // Plumb this in on the PUT side
END_REGION

REGION Network 7 (SCL): Error while sending CAN frames
   #TOF_SendError(IN:=#TESTUINT_SEND<>0,
                  PT:=T#10s);

   #TESTUINT_SEND := 0; //Reset Error

   //"WinCC_Alarm"(TriggerBit := #TOF_SendError.Q,
   //        Message := "DB_WinCCAlarms".Messages."3-Communication"."3002_ErrorWhileCANSending");
END_REGION

REGION Network 8 (SCL): Reset CAN module (queue)
   // This function resets the CAN-Module. For example sometimes the output queue for CAN-frames is full and sends an error. And the reset clears this queue, too.
   // Copied from process PLC
   IF "DB_Puma"."CAN-Reset_Required" THEN
       "Api_CtrlCAN_DB".sCtrl.fReq := True;
       "Api_CtrlCAN_DB".sCtrl.iFCN := 5;
       "DB_Puma"."CAN-Reset_Required" := FALSE;
   ELSIF "Api_CtrlCAN_DB".sCtrl.iFCN = 5 THEN

       "Api_CtrlCAN_DB".sCtrl.fReq := True;
       "Api_CtrlCAN_DB".sCtrl.iFCN := 1;
   END_IF;
END_REGION
END_FUNCTION_BLOCK

FUNCTION_BLOCK "CAN_CTRL"
{ S7_Optimized_Access := 'TRUE' }
VERSION : 0.1
   VAR_INPUT 
      HW_ID { ExternalAccessible := 'False'; ExternalVisible := 'False'; ExternalWritable := 'False'} : HW_IO;
      FCN { ExternalAccessible := 'False'; ExternalVisible := 'False'; ExternalWritable := 'False'} : Int;
      LEN_BufferLimit { ExternalAccessible := 'False'; ExternalVisible := 'False'; ExternalWritable := 'False'} : UInt;
      CANIdList : "FCN_1_CANIDList";
   END_VAR

   VAR_OUTPUT 
      BUSY { ExternalAccessible := 'False'; ExternalVisible := 'False'; ExternalWritable := 'False'} : Bool;
      RET { ExternalAccessible := 'False'; ExternalVisible := 'False'; ExternalWritable := 'False'} : UInt;
      CAN_STATUS { ExternalAccessible := 'False'; ExternalVisible := 'False'; ExternalWritable := 'False'} : Word;
   END_VAR

   VAR_IN_OUT 
      REQ { ExternalAccessible := 'False'; ExternalVisible := 'False'; ExternalWritable := 'False'} : Bool;
   END_VAR

   VAR 
      stat_siState : SInt := #cSTATE_INIT_CAN_CTRL;
      stat_fStartSFC : Bool := TRUE;
      stat_uiRetry : UInt := 0;
      stat_uiCmdLength : UInt := 0;
      stat_awRequest : Array[0..123] of Word;
      stat_abResponse : Array[0..247] of Byte;
      stat_RDREC {InstructionName := 'RDREC'; LibVersion := '1.0'} : RDREC;
      stat_WRREC {InstructionName := 'WRREC'; LibVersion := '1.1'} : WRREC;
   END_VAR

   VAR_TEMP 
      fBusy : Bool;
      fDoneValid : Bool;
      fError : Bool;
      dwStatus : DWord;
      wReturn : Word;
      uiResult : UInt;
      uiLen : UInt;
      udiCountElements : UDInt;
      iLoop : Int;
      iLoopEnd : Int;
   END_VAR

   VAR CONSTANT 
      cSTATE_INIT_CAN_CTRL : SInt := 0;
      cSTATE_WRITE_CAN_CTRL : SInt := 1;
      cSTATE_READ_CAN_CTRL : SInt := 2;
      cINDEX_CMD_CAN_CTRL : DInt := 16#9A;
      cMLEN_RDREC_CAN_CTRL : USInt := 248;
      cSRC_INDEX_CAN_CTRL : DInt := 0;
      cDEST_INDEX_CAN_CTRL : DInt := 2;
      cMAX_RETRY_CAN_CTRL : UInt := 1000;
      cMAX_NO_CANIDS_CAN_CTRL : UInt := 118;
   END_VAR


BEGIN
	(* ------------------------------------------------------------------------
	Title:        CAN_CTRL
	Description:  function processes the CAN_CTRL commands on a
	              CM CANopen module in transparent mode
	
	Inputs:       HW_ID:           hardware identifier of the CM module
	              FCN:             function code
	                               see manual: CAN_CTRL
	              LEN_BufferLimit: FCN: 1 <=> number if CAN ids to be transferred 
	                               FCN: 2 <=> value Buffer LIMIT REACHED
	              CANIdList:       points to the acceptance filter array
	                               - acceptance filter array:
	                                 - data type: Array[0..] of Word
	                                 - Array[0]: 1. CAN Id
	                                   Array[n]: (n + 1). CAN Id
	                                   bit 15: set     => receive
	                                           not set => remove
	
	InOut:        REQ:             TRUE : process CAN_CTRL
	                                      is automatically cleared when the command
	                                      has been processed
	                               FALSE: do not process CAN_CTRL
	                                      initializes the function
	                                           
	Outputs:      BUSY:            TRUE : function is running
	                               FALSE: function has been processed
	              RET:             result of the processed command
	                               only valid if output BUSY is FALSE
	                               see manual: RET ouput of CAN_CTRL 
	              CAN_STATUS:      CAN status:
	                               bit coded:
	                                 - bit  0 set: Bus off
	                                 - bit  1 set: error passive
	                                 - bit  2 set: receive queue: full
	                                 - bit  3 set: receive queue: half full
	                                 - bit  4 set: receive queue: warning limit reached
	                                 - bit  5 set: receive message lost
	                                 - bit  6 set: transmit queue: half full
	                                 - bit  7 set: transmit queue: warning limit reached
	                                 - bit 8 - 14: not used
	                                 - bit 15 set: valid
	                               CAN_STATUS is only valid if bit 15 is set:
	                               CAN_STATUS = 16#8000 <=> no error
	                               
	Hint:         - function needs minimum 2 calls before the response is available
	                  - delay time caused by the CM module:
	                    - time between reception and response: < 1ms
	                  - the more serious delay is caused by the asynchronous processing of
	                    the telegram whose transmission is requested by WRREC and RDREC
	              - the delay is not serious because it not blocking
	
	Author:       HMS
	Version:      1.0
	Date:         2017-03-19
	------------------------------------------------------------------------- *)
	
	// init Output RET
	#RET := 0;
	// init Output CAN_STATUS
	#CAN_STATUS := 0;
	
	IF #REQ = FALSE THEN
	    ///////////////////////////////////////////////////
	    // do not process CAN_CTRL
	    // initialize CAN_CTRL
	    ///////////////////////////////////////////////////    
	    #stat_siState := #cSTATE_INIT_CAN_CTRL;
	    #stat_uiRetry := 0;
	    #BUSY := FALSE;
	    RETURN;
	END_IF;
	
	// init Output BUSY
	#BUSY := TRUE;
	
	//==============================================================================  
	// main of "CAN_CTRL"()
	//==============================================================================  
	CASE #stat_siState OF
	        // initialize the data of the requested FCN command    
	    #cSTATE_INIT_CAN_CTRL:
	        GOTO CAN_CTRL_INIT_CMD;
	        
	        // transfer the command and its data to the CM module
	    #cSTATE_WRITE_CAN_CTRL:
	        GOTO CAN_CTRL_TRANSFER_CMD;
	        
	        // read result from the CM module
	    #cSTATE_READ_CAN_CTRL:
	        GOTO CAN_CTRL_GET_RESULT;
	        
	    ELSE
	        // state is not supported
	        // error code: state error (not defined in the manual)
	        #uiResult := 16#109F;
	        GOTO CAN_CTRL_DONE;
	END_CASE;
	
	//==============================================================================  
	// initialize the FCN specific data
	//==============================================================================  
	CAN_CTRL_INIT_CMD:
	
	// switch function code
	CASE #FCN OF
	    1:  // set acceptance filter in the module        
	        ///////////////////////////////////////////////////////////////////////////
	        // the CM module supports 2 types of "Set acceptance filter in the module"
	        // 1. #LEN_BufferLimit = 0
	        //      => disable all CAN-IDs
	        // 1. #LEN_BufferLimit > 0 
	        //      => selected CAN-IDs are entered in or removed from the acceptance
	        //         filter
	        //      => includes receive all CAN-IDs
	        ///////////////////////////////////////////////////////////////////////////
	        
	        ///////////////////////////////////////////////////////////////////////////
	        // #stat_awRequest[0]: FCN
	        // #stat_awRequest[1]: LEN
	        // #stat_awRequest[2...]: CAN Ids
	        ///////////////////////////////////////////////////////////////////////////
	
	        // function code: 
	        // - low address : function code
	        // - high address: 0 
	        #stat_awRequest[0] := 16#0100;
	        
	        // enter number of CAN-Ids:
	        // - big endian
	        #stat_awRequest[1] := UINT_TO_WORD(#LEN_BufferLimit);
	        
	        // number of data bytes to be written:
	        // - 4 bytes header + LEN_BufferLimit * 2
	        #stat_uiCmdLength := 4 + (#LEN_BufferLimit * 2);
	        
	        IF (#LEN_BufferLimit = 0) THEN
	            #stat_awRequest[2] := 16#0000;
	        ELSIF (#LEN_BufferLimit <= #cMAX_NO_CANIDS_CAN_CTRL) THEN
	            
	            // processing time MOVE_BLK:
	            // - CPU 1215C AC/DC/Rly needs
	            //       less than 0,240ms
	            //   to move 118 (maximum) CAN Ids            
	            MOVE_BLK(IN:=#CANIdList.FCN_1_CANIDList[#cSRC_INDEX_CAN_CTRL],
	                     COUNT:=#LEN_BufferLimit,
	                     OUT=>#stat_awRequest[#cDEST_INDEX_CAN_CTRL]);
	            
	            
	            // check if CAN-IDs are valid
	            // valid CAN-IDs
	            // - enable CAN ID : 16#xxxx OR 16#8000
	            //                   16#xxxx <= 16#7FF
	            // - enable all    : 16#FFFF 
	            // - disable CAN ID: 16#xxxx <= 16#7FF
	            #iLoopEnd := DINT_TO_INT(#cDEST_INDEX_CAN_CTRL) + UINT_TO_INT(#LEN_BufferLimit) - 1;
	            FOR #iLoop := DINT_TO_INT(#cDEST_INDEX_CAN_CTRL) TO #iLoopEnd DO
	                // Statement section FOR
	                IF (#stat_awRequest[#iLoop] AND 16#7FFF) > 16#7FF THEN
	                    IF #stat_awRequest[#iLoop] <> 16#FFFF THEN
	                        #uiResult := 16#109E;
	                        GOTO CAN_CTRL_DONE;
	                    END_IF;
	                END_IF;
	            END_FOR;
	                              
	        ELSE
	            // error code: too many CAN identifiers
	            #uiResult := 16#109C;
	            GOTO CAN_CTRL_DONE;
	        END_IF;
	        
	    2: // Set number of frames to store before warning (BUFFER LIMIT REACHED)
	        // default value of BUFFER LIMIT REACHED: 256
	        // 
	        // limitation:
	        //             1 <= BUFFER LIMIT REACHED value <= 256
	        IF ((#LEN_BufferLimit > 0) AND (#LEN_BufferLimit <= 256)) THEN
	            // - low address : function code
	            // - high address: 0
	            #stat_awRequest[0] := 16#0200;
	            
	            // enter buffer limit:
	            // - big endian
	            #stat_awRequest[1] := UINT_TO_WORD(#LEN_BufferLimit);
	            
	            // number of data bytes to be written:
	            // - 2 bytes header + 2 bytes data         
	            #stat_uiCmdLength := 4;
	        ELSE
	            // error code: buffer limit out of range
	            #uiResult := 16#109E;
	            GOTO CAN_CTRL_DONE;
	        END_IF;
	        
	    3: // Clear RX buffer
	        // - low address : function code
	        // - high address: 0
	        #stat_awRequest[0] := 16#0300;
	        
	        // no parameter / no data  
	        
	        // number of data bytes to be written:
	        // - 2 bytes header + 0 bytes data
	        #stat_uiCmdLength := 2;
	        
	    5: // Reset CAN controller (implies “Clear Bus Off”)
	        // - low address : function code
	        // - high address: 0
	        #stat_awRequest[0] := 16#0500;
	        
	        // no parameter / no data  
	        
	        // number of data bytes to be written:
	        // - 2 bytes header + 0 bytes data
	        #stat_uiCmdLength := 2;
	        
	    ELSE
	        // function code is not supported
	        // error code: "Function code (FCN) not allowed
	        #uiResult := 16#109B;
	        GOTO CAN_CTRL_DONE;
	END_CASE;
	
	// set start flag for SFC
	#stat_fStartSFC := TRUE;
	// init number of retry
	#stat_uiRetry := 0;
	// next state: transfer the command to the CM module
	#stat_siState := #cSTATE_WRITE_CAN_CTRL;
	
	
	//==============================================================================  
	// transfer the requested CAN control command to the CM module
	//==============================================================================  
	CAN_CTRL_TRANSFER_CMD:
	
	// download the requested command by using WRREC
	#stat_WRREC(REQ:=#stat_fStartSFC,
	           ID:=#HW_ID,
	           INDEX:=#cINDEX_CMD_CAN_CTRL,
	           LEN:=#stat_uiCmdLength,
	           DONE=>#fDoneValid,
	           BUSY=>#fBusy,
	           ERROR=>#fError,
	           STATUS=>#dwStatus,
	           RECORD:=#stat_awRequest);
	
	IF #fBusy = TRUE THEN
	    // reset variable to prevent WRREC to be triggered once more
	    #stat_fStartSFC := FALSE;
	    RETURN;
	ELSE
	    IF #fError = FALSE THEN
	        // seems no error occured, continue with read response
	        // init number of retry
	        #stat_uiRetry := 0;
	        
	        // set start flag for SFC
	        #stat_fStartSFC := TRUE;
	        
	        // next state:
	        // read the result from the CM module
	        #stat_siState := #cSTATE_READ_CAN_CTRL;
	    ELSE
	        //Write error
	        #wReturn := DWORD_TO_WORD(SHR(IN := #dwStatus, N := 8)) AND W#16#FFFF;
	        "SendReceiveErrorCode"(wReturn := #wReturn,
	                               bAddErrInfo := 16#00,
	                               uiErrorCode => #uiResult);
	        GOTO CAN_CTRL_DONE;
	    END_IF;
	END_IF;
	
	
	//==============================================================================  
	// read the result from the CM module
	//============================================================================== 
	CAN_CTRL_GET_RESULT:
	
	// upload the result by using RDREC
	#stat_RDREC(REQ:=#stat_fStartSFC,
	           ID:=#HW_ID,
	           INDEX:=#cINDEX_CMD_CAN_CTRL,
	           MLEN:=#cMLEN_RDREC_CAN_CTRL,
	           VALID=>#fDoneValid,
	           BUSY=>#fBusy,
	           ERROR=>#fError,
	           STATUS=>#dwStatus,
	           LEN=>#uiLen,
	           RECORD:=#stat_abResponse);
	
	IF #fBusy = TRUE THEN
	    // reset variable to prevent WRREC to be triggered once more
	    #stat_fStartSFC := FALSE;
	    RETURN;
	ELSE
	    #wReturn := DWORD_TO_WORD(SHR(IN := #dwStatus, N := 8)) AND W#16#FFFF;
	    
	    // check if
	    // - RDREC reports "DP slave or module not ready": 16#xx80B5xx
	    // - CM module repots "busy": 16#FE
	    IF (#wReturn = W#16#80B5) OR (#stat_abResponse[0] = w#16#FE) THEN
	        #stat_uiRetry := #stat_uiRetry + 1;
	        
	        IF #stat_uiRetry > #cMAX_RETRY_CAN_CTRL THEN
	            //Internal error  
	            #uiResult := 16#1013;
	            GOTO CAN_CTRL_DONE;
	        ELSE
	            // repeat: REQ input of RDREC must be set to TRUE
	            #stat_fStartSFC := TRUE;
	            RETURN;
	        END_IF;
	    ELSE
	        // check for failure 
	        IF #fError = TRUE THEN
	            // RDREC has reported a communication error
	            "SendReceiveErrorCode"(wReturn := #wReturn,
	                                   bAddErrInfo := 16#00,
	                                   uiErrorCode => #uiResult);
	        ELSIF #stat_abResponse[0] > 0 THEN
	            // command was rejected by the CM module
	            "SendReceiveErrorCode"(wReturn := 16#00FF,
	                                   bAddErrInfo := #stat_abResponse[0],
	                                   uiErrorCode => #uiResult);
	            // check if CAN status is available
	            IF #uiLen >= 2 THEN
	                #CAN_STATUS := BYTE_TO_WORD(#stat_abResponse[1]) OR 16#8000;
	            END_IF;
	        ELSE
	            // success
	            #uiResult := 0;
	            // check if CAN status is available
	            IF #uiLen >= 2 THEN
	                #CAN_STATUS := BYTE_TO_WORD(#stat_abResponse[1]) OR 16#8000;
	            END_IF;
	        END_IF; // IF #fError = TRUE THEN  ELSIF  ELSE
	    END_IF;   // IF (#wReturn = W#16#80B5) ... THEN  ELSE   
	    
	END_IF; // IF #fBusy = TRUE THEN ... ELSE
	
	
	//==============================================================================  
	// command has been processed
	//==============================================================================  
	CAN_CTRL_DONE:
	// initialize "CAN_CTRL"()
	#stat_siState := #cSTATE_INIT_CAN_CTRL;
	#stat_uiRetry := 0;
	
	// update outputs
	#RET := #uiResult;
	#BUSY := FALSE;
	
	// clear request at InOut
	#REQ := FALSE;
	
END_FUNCTION_BLOCK

FUNCTION "SendReceiveErrorCode" : Void
{ S7_Optimized_Access := 'TRUE' }
VERSION : 0.1
   VAR_INPUT 
      wReturn : Word;
      bAddErrInfo : Byte;
   END_VAR

   VAR_OUTPUT 
      uiErrorCode : UInt;
   END_VAR

   VAR_TEMP 
      wErrorCode : Word;
   END_VAR


BEGIN
	(* ------------------------------------------------------------------------
	Title:        SendReceiveErrorCode
	Description:  function calculates the error code according the manual of the
	              CM module for "CAN_CTRL"(), "CAN_RCV"(), "CAN_SEND"() and
	              "CAN_GET_DIAGNOSTIC"()
	
	Inputs:       wReturn:         raw error value
	              bAddErrInfo:     additional error info
	Outputs:      uiErrorCode      error code as described by the manual for
	                               the transparent CAN functions
	
	Author:       HMS
	Version:      1.0
	Date:         2014-08-20
	-------------------------------------------------------------------------*)
	IF #wReturn = W#16#8090 THEN
	  #uiErrorCode :=  16#3100;
	ELSIF #wReturn = W#16#8093 THEN
	  #uiErrorCode :=  16#3200;
	ELSIF #wReturn = W#16#80A0 OR #wReturn = W#16#80A1 THEN
	  #uiErrorCode :=  16#3300;
	ELSIF #wReturn = W#16#80A2 THEN
	  #uiErrorCode :=  16#3701;
	ELSIF #wReturn = W#16#80A3 THEN
	  #uiErrorCode :=  16#3600;
	ELSIF #wReturn = W#16#80A4 THEN
	  #uiErrorCode :=  16#3702;
	ELSIF #wReturn = W#16#80B2 THEN
	  #uiErrorCode :=  16#3400;
	ELSIF #wReturn = W#16#80B3 THEN
	  #uiErrorCode :=  16#3500;
	ELSIF #wReturn >= W#16#80C1 AND #wReturn <= W#16#80C6 THEN
	  #uiErrorCode :=  WORD_TO_UINT(#wReturn) - 16#80C0 + 16#3702;
	ELSIF #wReturn = 0 THEN
	  #uiErrorCode :=  16#3800 + BYTE_TO_UINT(#bAddErrInfo);
	ELSIF #wReturn = W#16#FF THEN
	  #uiErrorCode :=  16#3900 + BYTE_TO_UINT(#bAddErrInfo);
	ELSE
	  IF #wReturn <> 0 OR #bAddErrInfo = 0 THEN
	    #uiErrorCode :=  16#FF00;
	  ELSE
	    #uiErrorCode :=  BYTE_TO_UINT(SHL(IN:=#bAddErrInfo, N:=8));
	  END_IF;
	END_IF;
	
	
END_FUNCTION

FUNCTION_BLOCK "CAN_RCV"
{ S7_Optimized_Access := 'TRUE' }
VERSION : 0.1
   VAR_INPUT 
      REQ { ExternalAccessible := 'False'; ExternalVisible := 'False'; ExternalWritable := 'False'} : Bool;
      HW_ID { ExternalAccessible := 'False'; ExternalVisible := 'False'; ExternalWritable := 'False'} : HW_IO;
   END_VAR

   VAR_OUTPUT 
      BUSY { ExternalAccessible := 'False'; ExternalVisible := 'False'; ExternalWritable := 'False'} : Bool;
      RET { ExternalAccessible := 'False'; ExternalVisible := 'False'; ExternalWritable := 'False'} : UInt;
      CAN_STATUS { ExternalAccessible := 'False'; ExternalVisible := 'False'; ExternalWritable := 'False'} : Word;
      NO_FRAMES : SInt;
   END_VAR

   VAR_IN_OUT 
      CAN_FRAMES : "CANFrames";
   END_VAR

   VAR 
      stat_fStart : Bool := TRUE;
      stat_uiRetry : UInt := 0;
      stat_abResponse : Array[0..248] of Byte;
      stat_RDREC {InstructionName := 'RDREC'; LibVersion := '1.0'} : RDREC;
   END_VAR

   VAR_TEMP 
      fBusy : Bool;
      fValid : Bool;
      fError : Bool;
      dwStatus : DWord;
      uiLen : UInt;
      wReturn : Word;
      uiResult : UInt;
      iRetVal : Int;
   END_VAR

   VAR CONSTANT 
      cINDEX_CMD_CAN_RCV : DInt := 16#9B;
      cMLEN_RDREC_CAN_RCV : USInt := 248;
      cMAX_RETRY_CAN_RCV : UInt := 100;
      cMAX_NO_FRAMES_CAN_RCV : Byte := 19;
      cSRC_OFFSET_RESULT_CAN_RCV : DInt := 0;
      cSRC_OFFSET_CANSTATUS_MSB_CAN_RCV : DInt := 1;
      cSRC_OFFSET_CANSTATUS_LSB_CAN_RCV : DInt := 2;
      cSRC_OFFSET_NOFRAMES_CAN_RCV : DInt := 3;
      cSRC_OFFSET_DATA_CAN_RCV : DInt := 4;
      cDEST_INDEX_CAN_RCV : DInt := 0;
   END_VAR


BEGIN
	(* ------------------------------------------------------------------------
	Title:        CAN_RCV
	Description:  function uploads received CAN messages on a
	              CM CANopen module in transparent mode
	              maximum 19 messages are transferred per processed command
	              uploaded CAN frames are copied to the InOut parameter: CAN_FRAMES
	              
	Inputs:       REQ:             TRUE : process CAN_RCV
	                               FALSE: do not process CAN_RCV
	                                      initializes the function
	              HW_ID:           hardware identifier of the CM module
	              
	InOut:        CAN_FRAMES:      pointer to the destination area where to save the
	                               uploaded CAN frames
	
	Outputs:      BUSY:            TRUE : function is running
	                               FALSE: function has been processed: success or error
	              RET:             result of the processed command
	                               see description of output RET of CAN_RCV in the manual
	                               only valid if output BUSY is FALSE
	              CAN_STATUS:      CAN status:
	                               bit coded:
	                                 - bit  0 set: Bus off
	                                 - bit  1 set: error passive
	                                 - bit  2 set: receive queue: full
	                                 - bit  3 set: receive queue: half full
	                                 - bit  4 set: receive queue: warning limit reached
	                                 - bit  5 set: receive message lost
	                                 - bit  6 set: transmit queue: half full
	                                 - bit  7 set: transmit queue: warning limit reached
	                                 - bit 8 - 14: not used
	                                 - bit 15 set: valid
	                               CAN_STATUS is only valid if bit 15 is set:
	                               CAN_STATUS = 16#8000 <=> no error
	              NO_FRAMES:       number of uploaded CAN frames
	                               only valid if
	                                             output BUSY is FALSE
	                                             and output RET does not report an error 
	
	Hint:         - CAN messages must not be lost !!!
	                - function needs minimum 1 call before the response is available
	                  - delay time caused by the CM module:
	                    - time between reception and response: < 1ms
	                  - the more serious delay is caused by the asynchronous processing of
	                    the telegram whose transmission is requested by RDREC
	                    
	                - the frequency of the calls of "CAN_RCV"() is decisive !!!                     
	                - the frequency of the function call must guarantee that CAN
	                  frames are not lost
	
	
	Author:       HMS
	Version:      1.0
	Date:         2017-03-19
	------------------------------------------------------------------------- *)
	
	//==============================================================================
	// layout of the received byte stream:
	// - response of the accessed CM module to a CAN_RCV access
	//==============================================================================
	// - result reported by the CM module
	//     - stat_abResponse[0]
	// - CAN status
	//     - MSB <=> stat_abResponse[1]
	//     - LSB <=> stat_abResponse[2]
	//     only MSB transfers information
	// - number of uploaded CAN frames
	//     - stat_abResponse[3]
	// - uploaded CAN frames
	//     - stat_abResponse[4...]
	//       - each frames covers 12 bytes
	//           CAN-Id         : 2 bytes
	//           RTR            : 1 byte
	//           Data Size / DLC: 1 byte
	//           Data           : 8 bytes
	//       - 1. CAN frame
	//            stat_abResponse[4...15]
	//       - n. CAN frame
	//            stat_abResponse[4 + (n-1) * 12] ... stat_abResponse[4 + (n-1) * 12 + 15]
	
	//       maximum 19 CAN frames can be uploaded per processed CAN_RCV
	//==============================================================================
	
	//==============================================================================
	// init outputs
	// - to avoid misunderstanding
	//==============================================================================
	#RET := 0;
	#CAN_STATUS := 0;
	#NO_FRAMES := 0;
	
	//==============================================================================
	// check if command must be processed
	//==============================================================================
	IF #REQ = FALSE THEN
	    ///////////////////////////////////////////////////
	    // do not process CAN_RCV
	    // initialize CAN_RCV
	    ///////////////////////////////////////////////////
	    #stat_uiRetry := 0;
	    #stat_fStart := TRUE;
	    
	    #BUSY := FALSE;
	    RETURN;
	END_IF;
	
	// init Output #BUSY
	#BUSY := TRUE;
	
	//==============================================================================
	// upload CAN frames
	//==============================================================================
	// upload is done by RDREC
	#stat_RDREC(REQ:=#stat_fStart,
	            ID:=#HW_ID,
	            INDEX:=#cINDEX_CMD_CAN_RCV,
	            MLEN:=#cMLEN_RDREC_CAN_RCV,
	            VALID=>#fValid,
	            BUSY=>#fBusy,
	            ERROR=>#fError,
	            STATUS=>#dwStatus,
	            LEN=>#uiLen,
	            RECORD:=#stat_abResponse);
	
	IF #fBusy = TRUE THEN
	    // prevent RDREC to be triggered once more
	    #stat_fStart := FALSE;
	    RETURN;
	END_IF;
	
	//==============================================================================  
	// CAN_RCV command has been processed
	// check result
	//============================================================================== 
	#uiResult := 0;
	#wReturn := DWORD_TO_WORD(SHR(IN := #dwStatus, N := 8)) AND W#16#FFFF;
	
	////////////////////////////////////////////////////////////////
	// check if
	// - RDREC reports "DP slave or module not ready": 16#xx80B5xx
	// - CM module reports "busy": 16#FE
	//////////////////////////////////////////////////////////////// 
	IF (#wReturn = W#16#80B5) OR (#stat_abResponse[#cSRC_OFFSET_RESULT_CAN_RCV] = w#16#FE) THEN
	    #stat_uiRetry := #stat_uiRetry + 1;
	    IF #stat_uiRetry > #cMAX_RETRY_CAN_RCV THEN
	        //Internal error  
	        #uiResult := 16#1013;
	        GOTO CAN_RCV_DONE;
	    ELSE
	        // repeat: REQ input of RDREC must be set to TRUE
	        #stat_fStart := TRUE;
	        RETURN;
	    END_IF;
	ELSE // IF (#wReturn = W#16#80B5)...   
	    // check for failure 
	    IF #fError = TRUE THEN
	        // RDREC has reported a communication error
	        "SendReceiveErrorCode"(wReturn := #wReturn,
	                               bAddErrInfo := 16#00,
	                               uiErrorCode => #uiResult);
	        GOTO CAN_RCV_DONE;
	    ELSIF #stat_abResponse[#cSRC_OFFSET_RESULT_CAN_RCV] > 0 THEN
	        // command was rejected by the CM module
	        "SendReceiveErrorCode"(wReturn := 16#00FF,
	                               bAddErrInfo := #stat_abResponse[#cSRC_OFFSET_RESULT_CAN_RCV],
	                               uiErrorCode => #uiResult);
	        // check if CAN status is available
	        IF #uiLen >= 2 THEN
	            #CAN_STATUS := BYTE_TO_WORD(#stat_abResponse[#cSRC_OFFSET_CANSTATUS_MSB_CAN_RCV]) OR 16#8000;
	        END_IF;
	        GOTO CAN_RCV_DONE;
	    ELSE
	        // no failure is indicated
	        
	        // check if CAN status is available
	        IF #uiLen >= 2 THEN
	            #CAN_STATUS := BYTE_TO_WORD(#stat_abResponse[#cSRC_OFFSET_CANSTATUS_MSB_CAN_RCV]) OR 16#8000;
	        END_IF;
	        
	        // check number of frames in response
	        IF #stat_abResponse[#cSRC_OFFSET_NOFRAMES_CAN_RCV] = 0 THEN
	            // no CAN frames have been uploaded
	            GOTO CAN_RCV_DONE;
	        ELSIF #stat_abResponse[#cSRC_OFFSET_NOFRAMES_CAN_RCV] > #cMAX_NO_FRAMES_CAN_RCV THEN
	            // SW error: maximum 19 CAN frames can be uploaded
	            "SendReceiveErrorCode"(wReturn := 16#0000,
	                                   bAddErrInfo := #stat_abResponse[#cSRC_OFFSET_NOFRAMES_CAN_RCV],
	                                   uiErrorCode => #uiResult);
	            GOTO CAN_RCV_DONE;
	        ELSE
	            // CAN frames have been uploaded
	            GOTO UPDATE_UPLOADED_FRAMES;
	        END_IF;
	    END_IF; // IF #fError = TRUE THEN ELSIF ELSE 
	END_IF; // IF (#wReturn = W#16#80B5) ... THEN  ELSE   
	
	
	//==============================================================================  
	// copy uploaded CAN frames to the destination area
	//==============================================================================
	UPDATE_UPLOADED_FRAMES:
	
	
	IF (#stat_abResponse[#cSRC_OFFSET_NOFRAMES_CAN_RCV] > 0) AND (#stat_abResponse[#cSRC_OFFSET_NOFRAMES_CAN_RCV] <= 19) THEN
	    #NO_FRAMES := BYTE_TO_SINT(#stat_abResponse[#cSRC_OFFSET_NOFRAMES_CAN_RCV]);
	    MOVE_BLK(IN := #stat_abResponse[#cSRC_OFFSET_DATA_CAN_RCV],
	             COUNT := BYTE_TO_USINT(#stat_abResponse[#cSRC_OFFSET_NOFRAMES_CAN_RCV]) * 12,
	             OUT => #CAN_FRAMES.abCANFrames[#cDEST_INDEX_CAN_RCV]);
	    
	ELSE
	    #NO_FRAMES := 0;
	END_IF;
	
	
	//==============================================================================  
	// command has been processed
	//============================================================================== 
	CAN_RCV_DONE:
	// initialize "CAN_RCV"
	#stat_uiRetry := 0;
	#stat_fStart  := TRUE;
	#NO_FRAMES := BYTE_TO_SINT(#stat_abResponse[#cSRC_OFFSET_NOFRAMES_CAN_RCV]);
	
	#RET := #uiResult;
	#BUSY := FALSE;
	
END_FUNCTION_BLOCK

FUNCTION_BLOCK "CAN_SEND"
{ S7_Optimized_Access := 'TRUE' }
VERSION : 0.1
   VAR_INPUT 
      HW_ID { ExternalAccessible := 'False'; ExternalVisible := 'False'; ExternalWritable := 'False'} : HW_IO;
      NO_FRAMES : USInt;
      CAN_FRAMES : "CANFrames";
   END_VAR

   VAR_OUTPUT 
      BUSY { ExternalAccessible := 'False'; ExternalVisible := 'False'; ExternalWritable := 'False'} : Bool;
      RET { ExternalAccessible := 'False'; ExternalVisible := 'False'; ExternalWritable := 'False'} : UInt;
      CAN_STATUS { ExternalAccessible := 'False'; ExternalVisible := 'False'; ExternalWritable := 'False'} : Word;
   END_VAR

   VAR_IN_OUT 
      REQ { ExternalAccessible := 'False'; ExternalVisible := 'False'; ExternalWritable := 'False'} : Bool;
   END_VAR

   VAR 
      stat_siState : SInt := #cSTATE_INIT_CAN_SEND;
      stat_fStartSFC : Bool := TRUE;
      stat_usiNoFrames : USInt := 0;
      stat_uiRequestTotalSize : UInt := 0;
      stat_uiRetry : UInt := 0;
      stat_abRequest : Array[0..228] of Byte;
      stat_abResponse : Array[0..247] of Byte;
      stat_WRREC {InstructionName := 'WRREC'; LibVersion := '1.1'} : WRREC;
      stat_RDREC {InstructionName := 'RDREC'; LibVersion := '1.0'} : RDREC;
   END_VAR

   VAR_TEMP 
      fBusy : Bool;
      fDoneValid : Bool;
      fError : Bool;
      dwStatus : DWord;
      wReturn : Word;
      uiLen : UInt;
      iRetVal : Int;
      uiResult : UInt;
      diDataLoop : DInt;
      diDataLoopEnd : DInt;
      usiEntry_ByteString : USInt;
      usiOffset : USInt;
   END_VAR

   VAR CONSTANT 
      cSTATE_INIT_CAN_SEND : SInt := 0;
      cSTATE_WRITE_CAN_SEND : SInt := 1;
      cSTATE_READ_CAN_SEND : SInt := 2;
      cINDEX_CMD_CAN_SEND : DInt := 16#9C;
      cMLEN_RDREC_CAN_SEND : USInt := 248;
      cMAX_RETRY_CAN_SEND : UInt := 100;
      cMAX_NO_FRAMES_CAN_SEND : UInt := 19;
      cBYTE_SIZE_CAN_FRAME : USInt := 12;
      cOFFSET_CAN_FRAME_1 : USInt := 1;
      cOFFSET_DLC : USInt := 3;
   END_VAR


BEGIN
	(* ------------------------------------------------------------------------
	Title:        CAN_SEND
	Description:  function downloads CAN messages to the CM CANopen module
	              in transparent mode
	              maximum 19 messages can be transferred per processed command
	
	
	Inputs:       HW_ID:           hardware identifier of the CM module
	              NO_FRAMES:       number of CAN frames to be transferred
	              CAN_FRAMES:      source area where to get the CAN frames to be
	                               transmitted
	              
	InOut:        REQ:             TRUE : process CAN_SEND
	                                      is automatically cleared when the command
	                                      has been processed
	                               FALSE: do not process CAN_SEND
	                                      initializes the function
	
	Outputs:      BUSY:            TRUE : function is running
	                               FALSE: function has been processed: success or error
	              RESULT:          result of the processed command
	                               only valid if output BUSY is FALSE
	              CAN_STATUS:      CAN status:
	                               bit coded:
	                                 - bit  0 set: Bus off
	                                 - bit  1 set: error passive
	                                 - bit  2 set: receive queue: full
	                                 - bit  3 set: receive queue: half full
	                                 - bit  4 set: receive queue: warning limit reached
	                                 - bit  5 set: receive message lost
	                                 - bit  6 set: transmit queue: half full
	                                 - bit  7 set: transmit queue: warning limit reached
	                                 - bit 8 - 14: not used
	                                 - bit 15 set: valid
	                               CAN_STATUS is only valid if bit 15 is set:
	                               CAN_STATUS = 16#8000 <=> no error
	                               
	Hint:         - function needs minimum 2 calls before the response is available
	                  - delay time caused by the CM module:
	                    - time between reception and response: < 1ms
	                  - the more serious delay is caused by the asynchronous processing of
	                    the telegram whose transmission is requested by WRREC and RDREC
	              - cyclic transmission needs a good design by the application
	
	
	Author:       HMS
	Version:      1.0
	Date:         2017-03-19
	------------------------------------------------------------------------- *)
	
	// init Output RESULT
	#RET := 0;
	// init Output CAN_STATUS
	#CAN_STATUS := 0;
	
	IF #REQ = FALSE THEN
	    ///////////////////////////////////////////////////
	    // do not process CAN_SEND
	    // initialize CAN_SEND
	    /////////////////////////////////////////////////// 
	    #stat_uiRetry := 0;
	    #stat_siState := #cSTATE_INIT_CAN_SEND;
	    #BUSY := FALSE;
	    RETURN;
	END_IF;
	
	// init Output BUSY
	#BUSY := TRUE;
	
	
	//==============================================================================  
	// main of "CAN_SEND"()
	//==============================================================================  
	CASE #stat_siState OF
	    // initialize the data of the requested FCN command    
	    #cSTATE_INIT_CAN_SEND:
	        GOTO CAN_SEND_INIT;
	        
	    // transfer the command and its data to the CM module
	    #cSTATE_WRITE_CAN_SEND:
	        GOTO CAN_SEND_TRANSFER_CMD;
	        
	    // read result from the CM module
	    #cSTATE_READ_CAN_SEND:
	        GOTO CAN_SEND_GET_RESULT;
	        
	    ELSE
	        // state is not supported
	        // error code: state error (not defined in the manual)
	        #uiResult := 16#109F;
	        GOTO CAN_SEND_DONE;
	END_CASE;
	
	
	//==============================================================================  
	// initialize CAN_SEND command
	// - especially ask the application for CAN frames to be sent
	//==============================================================================
	CAN_SEND_INIT:
	
	// check number of CAN frames to be sent
	IF #NO_FRAMES = 0 THEN
	    GOTO CAN_SEND_DONE;
	END_IF;
	IF #NO_FRAMES > #cMAX_NO_FRAMES_CAN_SEND THEN
	    #uiResult := 16#109C;
	    GOTO CAN_SEND_DONE;
	END_IF;
	
	// copy CAN frames in byte array that is transferred to the CM module
	MOVE_BLK(IN:=#CAN_FRAMES.abCANFrames[0],
	         COUNT:=#NO_FRAMES * 12,
	         OUT=>#stat_abRequest[#cOFFSET_CAN_FRAME_1]);
	
	// check CAN frames if CAN-IDs and DLC are valid
	// - MSB of CAN-ID: (#cOFFSET_CAN_FRAME_1 + 0 )+ (n * #cBYTE_SIZE_CAN_FRAME); 0 <= n <= NO_FRAMES - 1
	// - LSB of CAN-ID: (#cOFFSET_CAN_FRAME_1 + 1) + (n * #cBYTE_SIZE_CAN_FRAME); 0 <= n <= NO_FRAMES - 1
	// - RTR:           (#cOFFSET_CAN_FRAME_1 + 2) + (n * #cBYTE_SIZE_CAN_FRAME); 0 <= n <= NO_FRAMES - 1
	// - DLC:           (#cOFFSET_CAN_FRAME_1 + 3) + (n * #cBYTE_SIZE_CAN_FRAME); 0 <= n <= NO_FRAMES - 1
	// - Data:          (#cOFFSET_CAN_FRAME_1 + 4...11) + (n * #cBYTE_SIZE_CAN_FRAME); 0 <= n <= NO_FRAMES - 1
	#usiOffset := #cOFFSET_CAN_FRAME_1;
	#diDataLoopEnd := USINT_TO_DINT(#NO_FRAMES) - 1;
	FOR #diDataLoop := 0 TO #diDataLoopEnd DO
	    // only MSB of the CAN-ID and DLC must be checked
	    IF     (#stat_abRequest[#usiOffset] > 16#07)
	        OR (#stat_abRequest[#usiOffset + #cOFFSET_DLC] > 16#08)
	    THEN
	        #uiResult := 16#109D;
	        GOTO CAN_SEND_DONE;
	    ELSE
	        #usiOffset := #usiOffset + #cBYTE_SIZE_CAN_FRAME;
	    END_IF;
	END_FOR;
	
	// update number of CAN frames to be sent and number of data to be transferred 
	#stat_abRequest[0] := USINT_TO_BYTE(#NO_FRAMES);
	#stat_uiRequestTotalSize := 1 + USINT_TO_UINT(#NO_FRAMES) * #cBYTE_SIZE_CAN_FRAME;
	
	// start write command
	#stat_uiRetry := 0;
	#stat_fStartSFC := TRUE;
	#stat_siState := #cSTATE_WRITE_CAN_SEND;
	
	
	//==============================================================================  
	// transfer the CAN frames to the CM module
	//==============================================================================
	CAN_SEND_TRANSFER_CMD:
	#stat_WRREC(REQ:=#stat_fStartSFC,
	            ID:=#HW_ID,
	            INDEX:=#cINDEX_CMD_CAN_SEND,
	            LEN:=#stat_uiRequestTotalSize,
	            DONE=>#fDoneValid,
	            BUSY=>#fBusy,
	            ERROR=>#fError,
	            STATUS=>#dwStatus,
	            RECORD:=#stat_abRequest);
	
	IF #fBusy = TRUE THEN
	    // reset variable to prevent WRREC to be triggered once more
	    #stat_fStartSFC := FALSE;
	    RETURN;
	ELSE
	    IF #fError = FALSE THEN
	        // seems no error occured, continue with read response
	        #stat_uiRetry := 0;
	        #stat_fStartSFC := TRUE;
	        #stat_siState := #cSTATE_READ_CAN_SEND;
	    ELSE
	        //Write error
	        #wReturn := DWORD_TO_WORD(SHR(IN := #dwStatus, N := 8)) AND W#16#FFFF;
	        "SendReceiveErrorCode"(wReturn := #wReturn,
	                               bAddErrInfo := 16#00,
	                               uiErrorCode => #uiResult);
	        GOTO CAN_SEND_DONE;
	    END_IF;
	END_IF; // IF #fBusy = FALSE THEN 
	
	
	//==============================================================================  
	// get the result from the CM module
	//==============================================================================
	CAN_SEND_GET_RESULT:
	#stat_RDREC(REQ:=#stat_fStartSFC,
	            ID:=#HW_ID,
	            INDEX:=#cINDEX_CMD_CAN_SEND,
	            MLEN:=#cMLEN_RDREC_CAN_SEND,
	            VALID=>#fDoneValid,
	            BUSY=>#fBusy,
	            ERROR=>#fError,
	            STATUS=>#dwStatus,
	            LEN=>#uiLen,
	            RECORD:=#stat_abResponse);
	
	IF #fBusy = TRUE THEN
	    // reset variable to prevent RDREC to be triggered once more
	    #stat_fStartSFC := FALSE;
	    RETURN;
	ELSE  
	      
	    #wReturn := DWORD_TO_WORD(SHR(IN:=#dwStatus,N:=8)) AND W#16#FFFF;
	
	    // check if
	    // - RDREC reports "DP slave or module not ready": 16#xx80B5xx
	    // - CM module repots "busy": 16#FE
	    IF (#wReturn = W#16#80B5) OR (#stat_abResponse[0] = w#16#FE) THEN
	        #stat_uiRetry := #stat_uiRetry + 1;
	        IF #stat_uiRetry > #cMAX_RETRY_CAN_SEND THEN
	            //Internal error  
	            #uiResult := 16#1013;
	            GOTO CAN_SEND_DONE;
	        ELSE
	            // repeat: REQ input of RDREC must be set to TRUE
	            #stat_fStartSFC := TRUE;
	            RETURN;
	        END_IF;
	    ELSE
	      // check for failure 
	      IF #fError = TRUE THEN
	          // RDREC has reported a communication error
	          "SendReceiveErrorCode"(wReturn:=#wReturn,
	                                 bAddErrInfo:=16#00,
	                                 uiErrorCode=>#uiResult);
	      ELSIF #stat_abResponse[0] > 0 THEN
	          // command was rejected by the CM module
	          "SendReceiveErrorCode"(wReturn:=16#00FF,
	                                 bAddErrInfo:=#stat_abResponse[0],
	                                 uiErrorCode=>#uiResult);
	          // check if CAN status is available
	          IF #uiLen >= 2 THEN
	              #CAN_STATUS := BYTE_TO_WORD(#stat_abResponse[1]) OR 16#8000;
	          END_IF;
	      ELSE
	          // success
	          #uiResult := 0;
	          // check if CAN status is available
	          IF #uiLen >= 2 THEN
	              #CAN_STATUS := BYTE_TO_WORD(#stat_abResponse[1]) OR 16#8000;
	          END_IF;
	      END_IF; // IF #fError = TRUE THEN  ELSIF  ELSE
	  END_IF;   // IF (#wReturn = W#16#80B5) ... THEN  ELSE   
	END_IF;     // IF #fBusy = TRUE ELSE THEN
	
	
	//==============================================================================  
	// command has been processed
	//==============================================================================
	CAN_SEND_DONE:
	// initialize "CAN_SEND"()    
	#stat_uiRetry := 0;
	#stat_siState := #cSTATE_INIT_CAN_SEND;
	
	// update outputs
	#RET := #uiResult;
	#BUSY := FALSE;
	
	// clear request at InOut
	#REQ := FALSE;
	
	
END_FUNCTION_BLOCK

ORGANIZATION_BLOCK "ModbusRTU"   // OB32, FBD, CyclicInterrupt
TITLE = Modbus RTU Communication
{ S7_Optimized_Access := 'TRUE' }
VERSION : 0.1
// Run the Modbus Master and place the fieldbus images into I/O memory
// stored: AutoNumber true, IsIECCheckEnabled false, SetENOAutomatically false
   VAR_INPUT
      Initial_Call : Bool;   // Initial call of this OB
      Event_Count : Int;   // Events discarded
   END_VAR
BEGIN

REGION Network 1
   // To enable communication, set bStart to TRUE
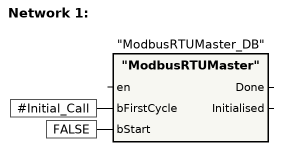
   "ModbusRTUMaster_DB"(bFirstCycle := #Initial_Call, bStart := FALSE);   // "ModbusRTUMaster"
END_REGION
END_ORGANIZATION_BLOCK

FUNCTION_BLOCK "ModbusRTUMaster"   // FB7, FBD
TITLE = Modbus RTU Master
{ S7_Optimized_Access := 'TRUE' }
VERSION : 0.1
// Sequence communication to several nodes. Each node is just added as more states to the state machine. There are better ways to do this but this will do for now.
// stored: AutoNumber true, IsIECCheckEnabled false, IsRetainMemResEnabled false, MemoryReserve 0, SetENOAutomatically false, UDAEnableTagReadback false
   VAR_INPUT
      bFirstCycle : Bool;
      bStart : Bool;
   END_VAR
   VAR_OUTPUT
      Done { ExternalAccessible := 'False'; ExternalVisible := 'False'; ExternalWritable := 'False'} : Bool;
      Initialised : Bool;   // 1 = successful init
   END_VAR
   VAR
      InitReq : Bool;
      InitErrorCode : Word;
      InitSuccess : Bool;
      ReadReq : Bool;
      MasterDoneStored : Bool;
      MasterStatus_stored : Word;
      MasterDone : Bool;
      MasterError : Bool;
      MasterBusy : Bool;
      MasterStatus : Word;
      State : USInt;
      Wait : TON_TIME;
      Node1CommCycles { S7_SetPoint := 'True'} : UDInt;
      Node2CommCycles : UDInt;
      Node10CommCycles : UDInt;
      Node20CommCycles : UDInt;
   END_VAR
   VAR_TEMP
      InitDone : Bool;
      InitError : Bool;
      InitStatus : Word;
   END_VAR
BEGIN

REGION Network 1 (SCL): Init modbus
   // NOTE: The DB at Modbus_Master's DATA_PTR pin must have "Optimized Access" disabled in its properties.
   // Modbus_Master's MODE input: (S7-1200 Programmable controller system manual, P. 1199 (A5E02486680-AM)
   // MODE 0 : Read Modbus address 1 to 9999, 10001 to 19999 as bits, 30001 to 39999, 40001 to 49999 as words
   // MODE 104 : Read Modbus address 0 to 65535 as words
   // Mode 1 : Write Modbus address 1 to 9999 as bits, 40001 to 49999 as words, 2 or more at a time
   // Mode 2 : As above but 1 or more at a time

   CASE #State OF
       0:  // IDLE
           IF #bStart = TRUE THEN
               #Done := FALSE;
               #InitReq := TRUE;
               #State := 1;
               #Node1CommCycles := 0;
               #Node2CommCycles := 0;
               #Node20CommCycles := 0;
           END_IF;
       1:  // INIT (runs once, not once every comm cycle)

           // For some reason, the duplex mode has to be set manually, and before the init block runs. 
           // Source: Siemens demo project for CM1241. Doesn't work without.
           "Modbus_Comm_Load_DB".MODE := 4;
           // REQ can only be high for one cycle. Wait 100ms (RESP_TO ) for slave response
           "Modbus_Comm_Load_DB"(REQ := #InitReq, 
                                 PORT := "Local~Modbus_RTU", 
                                 BAUD := 19200, 
                                 PARITY := 0, 
                                 FLOW_CTRL := 0, 
                                 RTS_ON_DLY := 0, 
                                 RTS_OFF_DLY := 0, 
                                 RESP_TO := 100, 
                                 MB_DB := "Modbus_Master_DB".MB_DB,
                                 DONE => #InitDone,
                                 ERROR => #InitError,
                                 STATUS => #InitStatus);
           #InitReq := FALSE;
           IF #InitDone THEN
               #InitSuccess := TRUE;
               #InitErrorCode := 0;
               #State := 4;
           ELSIF #InitError THEN
               #InitSuccess := FALSE;
               #InitErrorCode := #InitStatus;
               #State := 1;
           END_IF;
           #Initialised := #InitSuccess;
   (* ### Rewrite this for the actual nodes in the communication
       3: // Done
           // Optional wait between cycles
           //#Wait(IN := TRUE, PT := T#1ms);
           //IF #Wait.Q = TRUE THEN
           //    #Done := TRUE;
           //    #State := 4;
           //END_IF;
           #Done := TRUE;
           #State := 4;

       4: // Read Node 1
           "Modbus_Master_DB"(REQ := TRUE,
                               MB_ADDR := 1, 
                               MODE := 0, 
                               DATA_ADDR := 40009, 
                               DATA_LEN := 4,
                               DATA_PTR := P#DB10.DBX0.0 WORD 8,
                               DONE => #MasterDone,
                               BUSY => #MasterBusy,
                               ERROR => #MasterError,
                               STATUS => #MasterStatus);
           IF #MasterError = TRUE THEN 
               #MasterStatus_stored := #MasterStatus;
               "TA_State".%X0 := FALSE;
               #State := 6;
           ELSIF #MasterDone = TRUE THEN
               #MasterStatus := 0;
               "TA_State".%X0 := TRUE;
               "TA1_Rx".SW := "MasterData".dataPtr.data[0];
               "TA1_Rx".Act1 := "MasterData".dataPtr.data[1];
               "TA1_Rx".Act2 := "MasterData".dataPtr.data[2];
               "TA1_Rx".DataIO_12 := "MasterData".dataPtr.data[3];
               #State := 5;
           END_IF;
       5: // Write Node 1
           "MasterData".dataPtr.data[0] := "TA1_Tx".CW;
           "MasterData".dataPtr.data[1] := "TA1_Tx".Ref1;
           "MasterData".dataPtr.data[2] := "TA1_Tx".Ref2;
           "Modbus_Master_DB"(REQ := TRUE,
                               MB_ADDR := 1, 
                               MODE := 1, 
                               DATA_ADDR := 40001, 
                               DATA_LEN := 3,
                               DATA_PTR := P#DB10.DBX0.0 WORD 8,
                               DONE => #MasterDone,
                               BUSY => #MasterBusy,
                               ERROR => #MasterError,
                               STATUS => #MasterStatus);
           IF #MasterError = TRUE THEN 
               #MasterStatus_stored := #MasterStatus;
               "TA_State".%X0 := FALSE;
               #State := 6;
           ELSIF #MasterDone = TRUE THEN
               #MasterStatus := 0;
               "TA_State".%X0 := TRUE;
               #State := 6;
               #Node1CommCycles := #Node1CommCycles + 1;
           END_IF;
       6: // Read Node 2
           "Modbus_Master_DB"(REQ := TRUE,
                               MB_ADDR := 2, 
                               MODE := 0, 
                               DATA_ADDR := 40009, 
                               DATA_LEN := 4,
                               DATA_PTR := P#DB10.DBX0.0 WORD 8,
                               DONE => #MasterDone,
                               BUSY => #MasterBusy,
                               ERROR => #MasterError,
                               STATUS => #MasterStatus);
           IF #MasterError = TRUE THEN 
               #MasterStatus_stored := #MasterStatus;
               "TA_State".%X1 := FALSE;
               #State := 8;
           ELSIF #MasterDone = TRUE THEN
               #MasterStatus := 0;
               "TA_State".%X1 := TRUE;
               "TA2_Rx".SW :="MasterData".dataPtr.data[0];
               "TA2_Rx".Act1 := "MasterData".dataPtr.data[1];
               "TA2_Rx".Act2 := "MasterData".dataPtr.data[2];
               "TA2_Rx".DataIO_12 := "MasterData".dataPtr.data[3];
               #State := 7;
           END_IF;
       7: // Write Node 2
           "MasterData".dataPtr.data[0] := "TA2_Tx".CW;
           "MasterData".dataPtr.data[1] := "TA2_Tx".Ref1;
           "MasterData".dataPtr.data[2] := "TA2_Tx".Ref2;
           "Modbus_Master_DB"(REQ := TRUE,
                               MB_ADDR := 2, 
                               MODE := 1, 
                               DATA_ADDR := 40001, 
                               DATA_LEN := 3,
                               DATA_PTR := P#DB10.DBX0.0 WORD 8,
                               DONE => #MasterDone,
                               BUSY => #MasterBusy,
                               ERROR => #MasterError,
                               STATUS => #MasterStatus);
           IF #MasterError = TRUE THEN 
               #MasterStatus_stored := #MasterStatus;
               "TA_State".%X1 := FALSE;
               #State := 8;
           ELSIF #MasterDone = TRUE THEN
               #MasterStatus := 0;
               "TA_State".%X1 := TRUE;
               #State := 8;
               #Node2CommCycles := #Node2CommCycles + 1;   
           END_IF;

       8: // Read Node 10
           "Modbus_Master_DB"(REQ := TRUE,
                               MB_ADDR := 10, 
                               MODE := 0, 
                               DATA_ADDR := 40009, 
                               DATA_LEN := 4,
                               DATA_PTR := P#DB10.DBX0.0 WORD 8,
                               DONE => #MasterDone,
                               BUSY => #MasterBusy,
                               ERROR => #MasterError,
                               STATUS => #MasterStatus);
           IF #MasterError = TRUE THEN 
               #MasterStatus_stored := #MasterStatus;
               "TA_State".%X2 := FALSE;
               #State := 10;
           ELSIF #MasterDone = TRUE THEN
               #MasterStatus := 0;
               "TA_State".%X2 := TRUE;
               "TA10_Rx".SW :="MasterData".dataPtr.data[0];
               "TA10_Rx".Act1 := "MasterData".dataPtr.data[1];
               "TA10_Rx".Act2 := "MasterData".dataPtr.data[2];
               "TA10_Rx".DataIO_12 := "MasterData".dataPtr.data[3];
               #State := 9;
           END_IF;
       9: // Write Node 10
           "MasterData".dataPtr.data[0] := "TA10_Tx".CW;
           "MasterData".dataPtr.data[1] := "TA10_Tx".Ref1;
           "MasterData".dataPtr.data[2] := "TA10_Tx".Ref2;
           "Modbus_Master_DB"(REQ := TRUE,
                               MB_ADDR := 10, 
                               MODE := 1, 
                               DATA_ADDR := 40001, 
                               DATA_LEN := 3,
                               DATA_PTR := P#DB10.DBX0.0 WORD 8,
                               DONE => #MasterDone,
                               BUSY => #MasterBusy,
                               ERROR => #MasterError,
                               STATUS => #MasterStatus);
           IF #MasterError = TRUE THEN 
               #MasterStatus_stored := #MasterStatus;
               "TA_State".%X2 := FALSE;
               #State := 10;
           ELSIF #MasterDone = TRUE THEN
               "TA_State".%X2 := TRUE;
               #MasterStatus := 0;
               #State := 10;
               #Node10CommCycles := #Node10CommCycles + 1;   
           END_IF;

       10: // Read Node 20
           "Modbus_Master_DB"(REQ := TRUE,
                               MB_ADDR := 20, 
                               MODE := 104, 
                               DATA_ADDR := 16#0, 
                               DATA_LEN := 2,
                               DATA_PTR := P#DB10.DBX0.0 WORD 8,
                               DONE => #MasterDone,
                               BUSY => #MasterBusy,
                               ERROR => #MasterError,
                               STATUS => #MasterStatus);
           IF #MasterError = TRUE THEN 
               #MasterStatus_stored := #MasterStatus;
               "TA_State".%X7 := FALSE;
               #State := 3;
           ELSIF #MasterDone = TRUE THEN
               "TA_State".%X7 := TRUE;
               #MasterStatus := 0;
               "CVM1" := "MasterData".dataPtr.data[0];
               "CVM2" := "MasterData".dataPtr.data[1];
               #Node20CommCycles := #Node20CommCycles + 1;
               #State := 3;
           END_IF;

       // More nodes can go here, remember to jump to State 3 last.
   *)
   END_CASE;
END_REGION
END_FUNCTION_BLOCK

ORGANIZATION_BLOCK "S7_Comm"   // OB31, FBD, CyclicInterrupt
TITLE = Step 7 Communication with process control PLC
{ S7_Optimized_Access := 'TRUE' }
VERSION : 0.1
// stored: AutoNumber true, IsIECCheckEnabled false, SetENOAutomatically false
   VAR_INPUT
      Initial_Call : Bool;
      Event_Count : Int;
   END_VAR
BEGIN

REGION Network 1
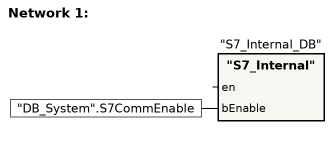
   "S7_Internal_DB"(bEnable := "DB_System".S7CommEnable);   // "S7_Internal"
END_REGION
END_ORGANIZATION_BLOCK

FUNCTION_BLOCK "S7_Internal"   // FB1, FBD
TITLE = Exchange data with Process PLC
{ S7_Optimized_Access := 'TRUE' }
VERSION : 0.1
// NOTES:
// 1. Size of CalcValue: 14 bytes
// 2. Max size one GET block can do: 222 bytes
// 3. Max. approx 10 simultaneous GET requests, so broken up into groups
// 4. Only one group is active per cycle. Total update cycle time is (Groups * OB31 cycle time)
// 5. REQ must stay high until the GET has completed (level signal). An edge on REQ will not work.
// 6. When a GET has completed it raises NDR for one cycle. The whole group is complete when all NDRs have been raised. GETs in the same group may not complete in the same cycle, so each NDR is used to SET a bit in xGroup to prevent retriggering while waiting (and thus getting stuck in that group as the NDRs will never go high at the same time). This is actually a sign that the OB cyclic rate is faster than the communication runs (two or more cycles per group) and that it should be increased, but at least it doesn't get stuck.
// 7. More groups can be added by following the model. WARNING: don't play here unless you are prepared for the consequences :-)
// stored: AutoNumber true, IsIECCheckEnabled false, IsRetainMemResEnabled false, MemoryReserve 100, SetENOAutomatically false, UDAEnableTagReadback false
   VAR_INPUT
      bEnable : Bool;   // 1 = do S7 comm, 0 = inhibit
   END_VAR
   VAR
      nGroup : USInt := 1;   // Read group
      xGroup1 : Byte;   // Group 1 read complete status bits
      xGroup2 : Byte;   // Group 2 read complete status bits
      xGroup3 : Byte;   // Group 3 read complete status bits
      xGroup4 : Byte;   // Group 4 read complete status bits
      GET_1 { S7_SetPoint := 'True'} : GET;
      GET_2 { S7_SetPoint := 'True'} : GET;
      GET_3 { S7_SetPoint := 'True'} : GET;
      GET_AI_4 { S7_SetPoint := 'True'} : GET;
      GET_AI_5 { S7_SetPoint := 'True'} : GET;
      GET_AI_6 { S7_SetPoint := 'True'} : GET;
      GET_AI_7 { S7_SetPoint := 'True'} : GET;
      GET_AI_8 { S7_SetPoint := 'True'} : GET;
      PUT_1 { S7_SetPoint := 'True'} : PUT;
      CommCycles { S7_SetPoint := 'True'} : UDInt;
      Group1Timeout : TON_TIME;
      Group2Timeout { S7_SetPoint := 'True'} : TON_TIME;
      Group3Timeout { S7_SetPoint := 'True'} : TON_TIME;
      Group4Timeout { S7_SetPoint := 'True'} : TON_TIME;
      RuntimeMemory { S7_SetPoint := 'True'} : LReal;
      RuntimeElapsed : LReal;   // How long one comm cycle takes
   END_VAR
   VAR_TEMP
      Group1Done : Bool;
      Group2Done : Bool;
      Group3Done : Bool;
      Group4Done : Bool;
   END_VAR
   VAR CONSTANT
      GroupTimeout : Time := T#3s;
   END_VAR
   VAR_TEMP   // added for the SCL form of the ladder/FBD networks
      _w1 : Bool;
   END_VAR
BEGIN

REGION Network 1: Group 1: GET
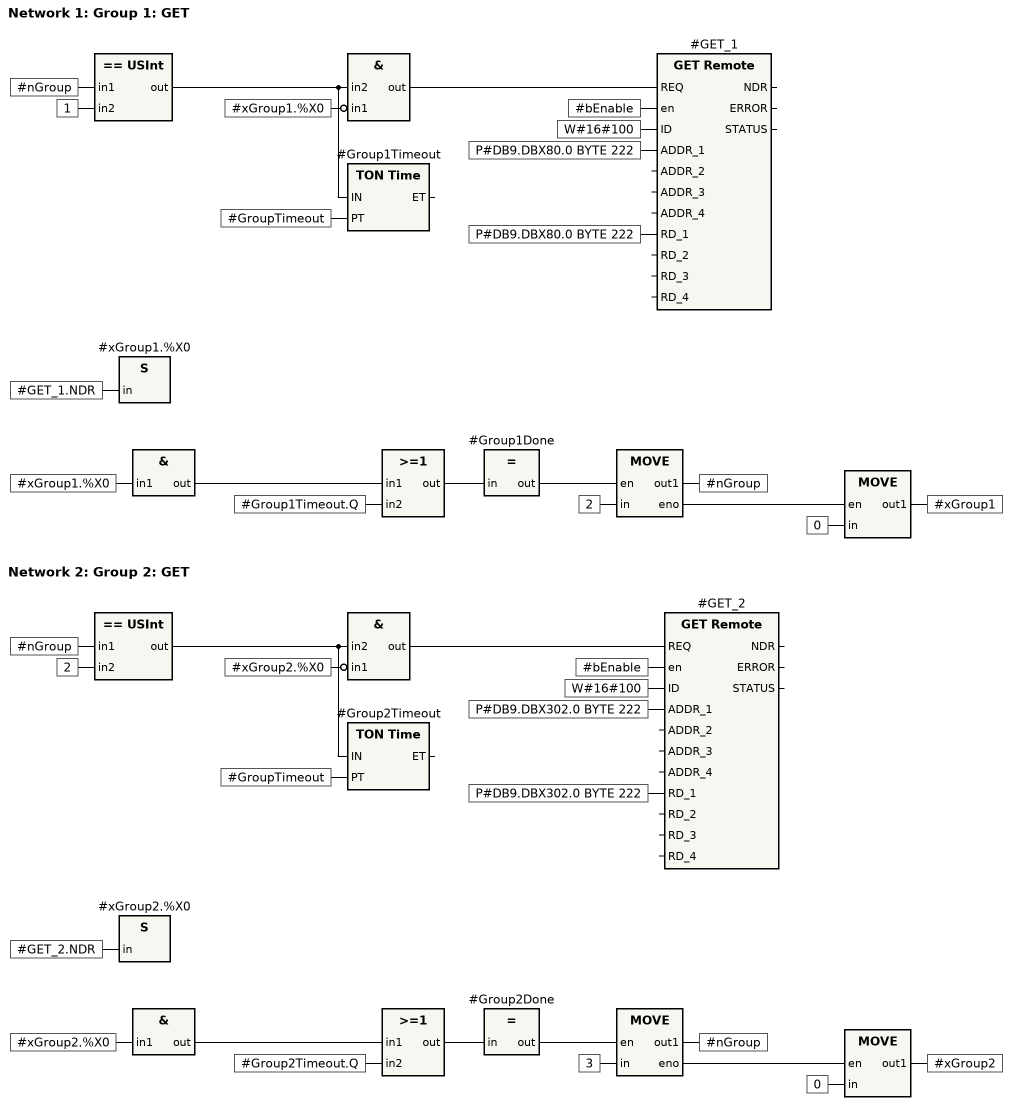
   #_w1 := #nGroup = 1;
   IF #bEnable THEN
       #GET_1(REQ := #_w1 AND NOT #xGroup1.%X0,   // GET
              ID := W#16#100,
              ADDR_1 := P#DB9.DBX80.0 BYTE 222,
              RD_1 := P#DB9.DBX80.0 BYTE 222);
   END_IF;
   #Group1Timeout(IN := #_w1, PT := #GroupTimeout);   // TON
   IF #GET_1.NDR THEN #xGroup1.%X0 := TRUE; END_IF;
   #Group1Done := #xGroup1.%X0 OR #Group1Timeout.Q;
   IF #Group1Done THEN
       #nGroup := 2;
       #xGroup1 := 0;
   END_IF;
END_REGION

REGION Network 2: Group 2: GET
   #_w1 := #nGroup = 2;
   IF #bEnable THEN
       #GET_2(REQ := #_w1 AND NOT #xGroup2.%X0,   // GET
              ID := W#16#100,
              ADDR_1 := P#DB9.DBX302.0 BYTE 222,
              RD_1 := P#DB9.DBX302.0 BYTE 222);
   END_IF;
   #Group2Timeout(IN := #_w1, PT := #GroupTimeout);   // TON
   IF #GET_2.NDR THEN #xGroup2.%X0 := TRUE; END_IF;
   #Group2Done := #xGroup2.%X0 OR #Group2Timeout.Q;
   IF #Group2Done THEN
       #nGroup := 3;
       #xGroup2 := 0;
   END_IF;
END_REGION

REGION Network 3: Group 3: GET
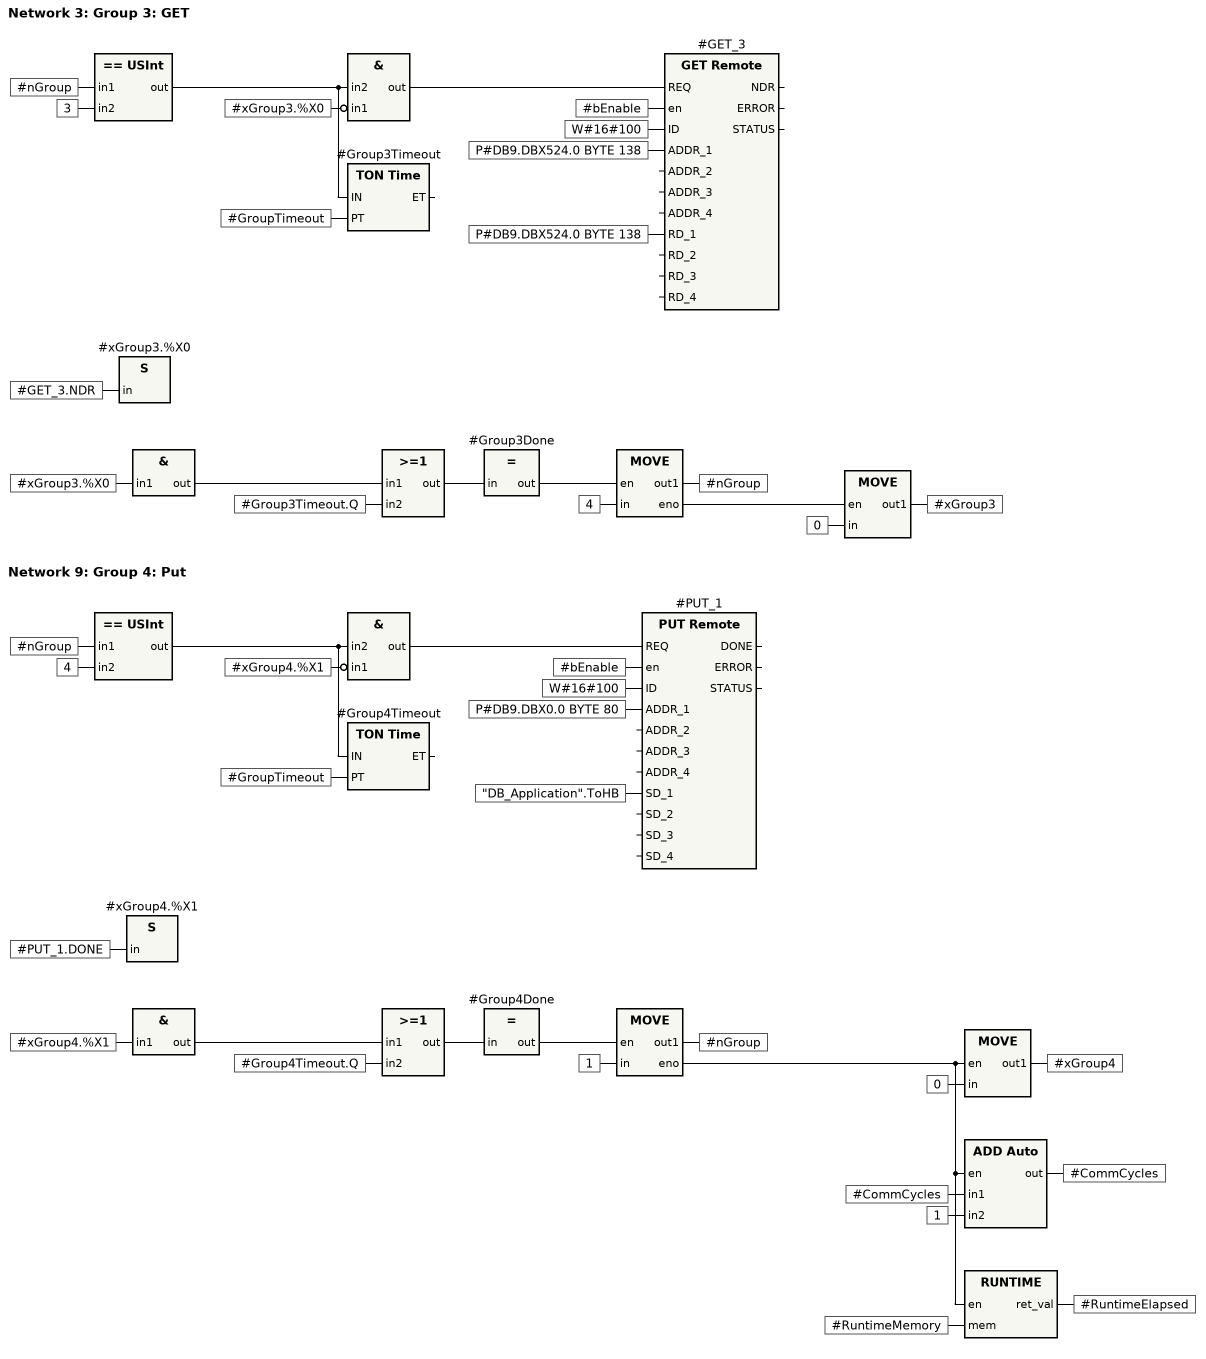
   #_w1 := #nGroup = 3;
   IF #bEnable THEN
       #GET_3(REQ := #_w1 AND NOT #xGroup3.%X0,   // GET
              ID := W#16#100,
              ADDR_1 := P#DB9.DBX524.0 BYTE 138,
              RD_1 := P#DB9.DBX524.0 BYTE 138);
   END_IF;
   #Group3Timeout(IN := #_w1, PT := #GroupTimeout);   // TON
   IF #GET_3.NDR THEN #xGroup3.%X0 := TRUE; END_IF;
   #Group3Done := #xGroup3.%X0 OR #Group3Timeout.Q;
   IF #Group3Done THEN
       #nGroup := 4;
       #xGroup3 := 0;
   END_IF;
END_REGION

REGION Network 4 (SCL): DB_AI
   // Update on new value
   IF #Group3Done = TRUE THEN
       "DB_Heatbooster".AI.HBL_TT_502.fValue := "DB_Application".FromHB.DB_AI.HBL_TT_502;
       "DB_Heatbooster".AI.HBL_PT_503.fValue := "DB_Application".FromHB.DB_AI.HBL_PT_503;
       "DB_Heatbooster".AI.HBL_TT_504.fValue := "DB_Application".FromHB.DB_AI.HBL_TT_504;
       "DB_Heatbooster".AI.HBL_LT_510.fValue := "DB_Application".FromHB.DB_AI.HBL_LT_510;
       "DB_Heatbooster".AI.HBL_PT_511.fValue := "DB_Application".FromHB.DB_AI.HBL_PT_511;
       "DB_Heatbooster".AI.HBL_TT_512.fValue := "DB_Application".FromHB.DB_AI.HBL_TT_512;
       "DB_Heatbooster".AI.HBL_TT_516.fValue := "DB_Application".FromHB.DB_AI.HBL_TT_516;
       "DB_Heatbooster".AI.HBL_PT_517.fValue := "DB_Application".FromHB.DB_AI.HBL_PT_517;
       "DB_Heatbooster".AI.HBL_TT_518.fValue := "DB_Application".FromHB.DB_AI.HBL_TT_518;
       "DB_Heatbooster".AI.HBL_PT_519.fValue := "DB_Application".FromHB.DB_AI.HBL_PT_519;
       "DB_Heatbooster".AI.HBL_FT_520.fValue := "DB_Application".FromHB.DB_AI.HBL_FT_520;
       "DB_Heatbooster".AI.HBL_TT_530.fValue := "DB_Application".FromHB.DB_AI.HBL_TT_530;
       "DB_Heatbooster".AI.HBL_PT_531.fValue := "DB_Application".FromHB.DB_AI.HBL_PT_531;
       "DB_Heatbooster".AI.HBL_TT_532.fValue := "DB_Application".FromHB.DB_AI.HBL_TT_532;
       "DB_Heatbooster".AI.HBL_TT_533.fValue := "DB_Application".FromHB.DB_AI.HBL_TT_533;
       "DB_Heatbooster".AI.HBL_PT_534.fValue := "DB_Application".FromHB.DB_AI.HBL_PT_534;
       "DB_Heatbooster".AI.HBL_AT_535.fValue := "DB_Application".FromHB.DB_AI.HBL_AT_535;
       "DB_Heatbooster".AI.HBL_TT_540.fValue := "DB_Application".FromHB.DB_AI.HBL_TT_540;
       "DB_Heatbooster".AI.HBL_PT_541.fValue := "DB_Application".FromHB.DB_AI.HBL_PT_541;
       "DB_Heatbooster".AI.HBL_TT_542.fValue := "DB_Application".FromHB.DB_AI.HBL_TT_542;
       "DB_Heatbooster".AI.HBL_TT_543.fValue := "DB_Application".FromHB.DB_AI.HBL_TT_543;
       "DB_Heatbooster".AI.HBL_PT_544.fValue := "DB_Application".FromHB.DB_AI.HBL_PT_544;
       "DB_Heatbooster".AI.HBL_AT_545.fValue := "DB_Application".FromHB.DB_AI.HBL_AT_545;
       "DB_Heatbooster".AI.HBL_TT_546.fValue := "DB_Application".FromHB.DB_AI.HBL_TT_546;
       "DB_Heatbooster".AI.HBL_PT_547.fValue := "DB_Application".FromHB.DB_AI.HBL_PT_547;
       "DB_Heatbooster".AI.HBL_TT_571.fValue := "DB_Application".FromHB.DB_AI.HBL_TT_571;
       "DB_Heatbooster".AI.HBL_PT_572.fValue := "DB_Application".FromHB.DB_AI.HBL_PT_572;
       "DB_Heatbooster".AI.HBL_TT_573.fValue := "DB_Application".FromHB.DB_AI.HBL_TT_573;
       "DB_Heatbooster".AI.HBL_LT_610.fValue := "DB_Application".FromHB.DB_AI.HBL_LT_610;
       "DB_Heatbooster".AI.HBL_TT_611.fValue := "DB_Application".FromHB.DB_AI.HBL_TT_611;
       "DB_Heatbooster".AI.HBL_PT_612.fValue := "DB_Application".FromHB.DB_AI.HBL_PT_612;
       "DB_Heatbooster".AI.HBL_CT_615.fValue := "DB_Application".FromHB.DB_AI.HBL_CT_615;
       "DB_Heatbooster".AI.HBL_PT_618.fValue := "DB_Application".FromHB.DB_AI.HBL_PT_618;
       "DB_Heatbooster".AI.HBL_PT_635.fValue := "DB_Application".FromHB.DB_AI.HBL_PT_635;
       "DB_Heatbooster".AI.HBL_PT_636.fValue := "DB_Application".FromHB.DB_AI.HBL_PT_636;
       "DB_Heatbooster".AI.HBL_LT_650.fValue := "DB_Application".FromHB.DB_AI.HBL_LT_650;
       "DB_Heatbooster".AI.HBL_PT_651.fValue := "DB_Application".FromHB.DB_AI.HBL_PT_651;
       "DB_Heatbooster".AI.HBL_PT_701.fValue := "DB_Application".FromHB.DB_AI.HBL_PT_701;
       "DB_Heatbooster".AI.HBL_PT_702.fValue := "DB_Application".FromHB.DB_AI.HBL_PT_702;
       "DB_Heatbooster".AI.HBL_PT_703.fValue := "DB_Application".FromHB.DB_AI.HBL_PT_703;
       "DB_Heatbooster".AI.CPC_LT_870.fValue := "DB_Application".FromHB.DB_AI.CPC_LT_870;
       "DB_Heatbooster".AI.CPC_TT_871.fValue := "DB_Application".FromHB.DB_AI.CPC_TT_871;
       "DB_Heatbooster".AI.CPC_PT_872.fValue := "DB_Application".FromHB.DB_AI.CPC_PT_872;
       "DB_Heatbooster".AI.CPC_PT_862.fValue := "DB_Application".FromHB.DB_AI.CPC_PT_862;
       "DB_Heatbooster".AI.HBL_TT_901.fValue := "DB_Application".FromHB.DB_AI.HBL_TT_901;
       "DB_Heatbooster".AI.HBL_PT_902.fValue := "DB_Application".FromHB.DB_AI.HBL_PT_902;

